//Balança de sólido 2
//Calculo peso com erro superior
PESO_ERRO_MAX_BLS2 := PRST_PESO_BLS2 + (PRST_PESO_BLS2 * (PRST_PORCENTAGEM_ERRO_PESO_BLS2 / 100));
//compara a banda
IF LEITURA_PESO_BLS2 > PESO_ERRO_MAX_BLS2 AND PRST_PESO_BLS2 > 0 AND BLS2_CARREGADA = TRUE AND BTS_PERMI_DESCAR_PESO_MAX_BLS2 = FALSE THEN
	AL_PESO_ALTO_BLS2 := TRUE;
ELSIF BTS_PERMI_DESCAR_PESO_MAX_BLS2 = TRUE OR PRST_PESO_BLS2 = 0 THEN	
	AL_PESO_ALTO_BLS2 := FALSE;	
END_IF

//Balança de sólido 3
//Calculo peso com erro superior
PESO_ERRO_MAX_BLS3 := PRST_PESO_BLS3 + (PRST_PESO_BLS3 * (PRST_PORCENTAGEM_ERRO_PESO_BLS3 / 100));
//compara a banda
IF LEITURA_PESO_BLS3 > PESO_ERRO_MAX_BLS3 AND PRST_PESO_BLS3 > 0 AND BLS3_CARREGADA = TRUE AND BTS_PERMI_DESCAR_PESO_MAX_BLS3 = FALSE THEN
	AL_PESO_ALTO_BLS3 := TRUE;
ELSIF BTS_PERMI_DESCAR_PESO_MAX_BLS3 = TRUE OR PRST_PESO_BLS3 = 0 THEN	
	AL_PESO_ALTO_BLS3 := FALSE;	
END_IF

//Balança de sólido 4
//Calculo peso com erro superior
PESO_ERRO_MAX_BLS4 := PRST_PESO_BLS4 + (PRST_PESO_BLS4 * (PRST_PORCENTAGEM_ERRO_PESO_BLS4 / 100));
//compara a banda
IF LEITURA_PESO_BLS4 > PESO_ERRO_MAX_BLS4 AND PRST_PESO_BLS4 > 0 AND BLS4_CARREGADA = TRUE AND BTS_PERMI_DESCAR_PESO_MAX_BLS4 = FALSE THEN
	AL_PESO_ALTO_BLS4 := TRUE;
ELSIF BTS_PERMI_DESCAR_PESO_MAX_BLS4 = TRUE OR PRST_PESO_BLS4 = 0 THEN	
	AL_PESO_ALTO_BLS4 := FALSE;	
END_IF

//Balança de sólido 5
//Calculo peso com erro superior
PESO_ERRO_MAX_BLS5 := PRST_PESO_BLS5 + (PRST_PESO_BLS5 * (PRST_PORCENTAGEM_ERRO_PESO_BLS5 / 100));
//compara a banda
IF LEITURA_PESO_BLS5 > PESO_ERRO_MAX_BLS5 AND PRST_PESO_BLS5 > 0 AND BLS5_CARREGADA = TRUE AND BTS_PERMI_DESCAR_PESO_MAX_BLS5 = FALSE THEN
	AL_PESO_ALTO_BLS5 := TRUE;
ELSIF BTS_PERMI_DESCAR_PESO_MAX_BLS5 = TRUE OR PRST_PESO_BLS5 = 0 THEN	
	AL_PESO_ALTO_BLS5 := FALSE;	
END_IF

//Balança de liquido 1
//Calculo peso com erro superior
PESO_ERRO_MAX_BLL1 := PRST_PESO_BLL1 + (PRST_PESO_BLL1 * (PRST_PORCENTAGEM_ERRO_PESO_BLL1 / 100));
//compara a banda
IF LEITURA_PESO_BLL1 > PESO_ERRO_MAX_BLL1 AND PRST_PESO_BLL1 > 0 AND BLL1_CARREGADA = TRUE AND BTS_PERMI_DESCAR_PESO_MAX_BLL1 = FALSE THEN
	AL_PESO_ALTO_BLL1 := TRUE;
ELSIF BTS_PERMI_DESCAR_PESO_MAX_BLL1 = TRUE OR PRST_PESO_BLL1 = 0 THEN	
	AL_PESO_ALTO_BLL1 := FALSE;	
END_IF

//Balança de liquido 2
//Calculo peso com erro superior
PESO_ERRO_MAX_BLL2 := PRST_PESO_BLL2 + (PRST_PESO_BLL2 * (PRST_PORCENTAGEM_ERRO_PESO_BLL2 / 100));
//compara a banda
IF LEITURA_PESO_BLL2 > PESO_ERRO_MAX_BLL2 AND PRST_PESO_BLL2 > 0 AND BLL2_CARREGADA = TRUE AND BTS_PERMI_DESCAR_PESO_MAX_BLL2 = FALSE THEN
	AL_PESO_ALTO_BLL2 := TRUE;
ELSIF BTS_PERMI_DESCAR_PESO_MAX_BLL2 = TRUE OR PRST_PESO_BLL2 = 0  THEN	
	AL_PESO_ALTO_BLL2 := FALSE;	
END_IF

//Balança de liquido 3
//Calculo peso com erro superior
PESO_ERRO_MAX_BLL3 := PRST_PESO_BLL3 + (PRST_PESO_BLL3 * (PRST_PORCENTAGEM_ERRO_PESO_BLL3 / 100));
//compara a banda
IF LEITURA_PESO_BLL3 > PESO_ERRO_MAX_BLL3 AND PRST_PESO_BLL3 > 0 AND BLL3_CARREGADA = TRUE AND BTS_PERMI_DESCAR_PESO_MAX_BLL3 = FALSE THEN
	AL_PESO_ALTO_BLL3 := TRUE;
ELSIF BTS_PERMI_DESCAR_PESO_MAX_BLL3 = TRUE OR PRST_PESO_BLL3 = 0  THEN	
	AL_PESO_ALTO_BLL3 := FALSE;	
END_IF

//Balança de liquido 4
//Calculo peso com erro superior
PESO_ERRO_MAX_BLL4 := PRST_PESO_BLL4 + (PRST_PESO_BLL4 * (PRST_PORCENTAGEM_ERRO_PESO_BLL4 / 100));
//compara a banda
IF LEITURA_PESO_BLL4 > PESO_ERRO_MAX_BLL4 AND PRST_PESO_BLL4 > 0 AND BLL4_CARREGADA = TRUE AND BTS_PERMI_DESCAR_PESO_MAX_BLL4 = FALSE THEN
	AL_PESO_ALTO_BLL4 := TRUE;
ELSIF BTS_PERMI_DESCAR_PESO_MAX_BLL4 = TRUE OR PRST_PESO_BLL4 = 0  THEN	
	AL_PESO_ALTO_BLL4 := FALSE;
END_IF

//======================= Exaustores =========================================================

//Alame estrela Exaustor FM2 

IF SD_EXFM2_E = TRUE AND (ED_CFEXFM2_P = FALSE AND ED_CFEXFM2_E = FALSE) THEN
	LIBERA_TEMPO_AL_FM2E:= TRUE;
ELSE
	LIBERA_TEMPO_AL_FM2E:= FALSE;
END_IF

TMR_TEMPO_ALARME_FM2_E(IN:= LIBERA_TEMPO_AL_FM2E, PT:= T#6S);

IF TMR_TEMPO_ALARME_FM2_E.Q = TRUE THEN
	AL_EXFM2_E:=TRUE;
END_IF

//Alame triangulo Exaustor FM2 

IF SD_EXFM2_T = TRUE AND (ED_CFEXFM2_P = FALSE AND ED_CFEXFM2_T = FALSE) THEN
	LIBERA_TEMPO_AL_FM2T:= TRUE;
ELSE
	LIBERA_TEMPO_AL_FM2T:= FALSE;
END_IF

TMR_TEMPO_ALARME_FM2_T(IN:= LIBERA_TEMPO_AL_FM2T, PT:= T#6S);

IF TMR_TEMPO_ALARME_FM2_T.Q = TRUE THEN
	AL_EXFM2_T:=TRUE;
END_IF

//Alame estrela Ventilador FM2 

IF SD_VEXFM2_E = TRUE AND (ED_CFVEXFM2_P = FALSE AND ED_CFVEXFM2_E = FALSE) THEN
	LIBERA_TEMPO_AL_VFM2E:= TRUE;
ELSE
	LIBERA_TEMPO_AL_VFM2E:= FALSE;
END_IF

TMR_TEMPO_ALARME_VFM2_E(IN:= LIBERA_TEMPO_AL_VFM2E, PT:= T#6S);

IF TMR_TEMPO_ALARME_VFM2_E.Q = TRUE THEN
	AL_VEXFM2_E:=TRUE;
END_IF

//Alame triangulo Ventilador FM2 

IF SD_VEXFM2_T = TRUE AND (ED_CFVEXFM2_P = FALSE AND ED_CFVEXFM2_T = FALSE) THEN
	LIBERA_TEMPO_AL_VFM2T:= TRUE;
ELSE
	LIBERA_TEMPO_AL_VFM2T:= FALSE;
END_IF

TMR_TEMPO_ALARME_VFM2_T(IN:= LIBERA_TEMPO_AL_VFM2T, PT:= T#6S);

IF TMR_TEMPO_ALARME_VFM2_T.Q = TRUE THEN
	AL_VEXFM2_T:=TRUE;
END_IF

//Alarme Exautor da torre (125 cv) 

IF ED_EX125_ALAR = TRUE THEN
	AL_EXTORRE:= TRUE;
END_IF


//Alarme ventilador do queimador (100 cv) 

IF ED_EX100_ALAR = TRUE THEN
	AL_VENTQUEIMADOR:= TRUE;
END_IF

//=============================== Bombas ============================================

//Alarme falta oleo bomba de alimentação 

IF SD_BAO = TRUE AND ED_NVBO = FALSE THEN
	LIBERA_TEMPO_AL_BALIOLEO := TRUE;
ELSE
	LIBERA_TEMPO_AL_BALIOLEO := FALSE;
END_IF

TMR_TEMPO_ALARME_BOMBA_ALIM_OLEO(IN:=LIBERA_TEMPO_AL_BALIOLEO, PT:=T#20S);

IF TMR_TEMPO_ALARME_BOMBA_ALIM_OLEO.Q = TRUE THEN
	AL_BOCOMBFALT := TRUE;
END_IF


//Bomba de Blend 
IF SD_BBD = TRUE AND ED_BB_D = FALSE THEN
	LIBERA_TEMPO_AL_BBBLEND:=TRUE;
ELSE
	LIBERA_TEMPO_AL_BBBLEND:= FALSE;
END_IF

TMR_TEMPO_ALARME_BBBLEND(IN:=LIBERA_TEMPO_AL_BBBLEND, PT:=T#15S);

IF TMR_TEMPO_ALARME_BBBLEND.Q = TRUE THEN
	AL_BBLEND:=TRUE;
END_IF


//Bomba de Silicato (Acrilato) 
IF SD_BSIL = TRUE AND ED_BSI_D = FALSE THEN
	LIBERA_TEMPO_AL_BBSILICATO:=TRUE;
ELSE
	LIBERA_TEMPO_AL_BBSILICATO:= FALSE;
END_IF

TMR_TEMPO_ALARME_BBSILICATO(IN:=LIBERA_TEMPO_AL_BBSILICATO, PT:=T#15S);

IF TMR_TEMPO_ALARME_BBSILICATO.Q = TRUE THEN
	AL_SILI:=TRUE;
END_IF


//Bomba de Sulfonico 
IF SD_BSUL = TRUE AND ED_BSU_D = FALSE THEN
	LIBERA_TEMPO_AL_BBSULFONICO:=TRUE;
ELSE
	LIBERA_TEMPO_AL_BBSULFONICO:= FALSE;
END_IF

TMR_TEMPO_ALARME_BBSULFONICO(IN:=LIBERA_TEMPO_AL_BBSULFONICO, PT:=T#15S);

IF TMR_TEMPO_ALARME_BBSULFONICO.Q = TRUE THEN
	AL_BBSULFONICO:=TRUE;
END_IF


//Bomba de Agua 
IF SD_BAG = TRUE AND ED_BA_D = FALSE THEN
	LIBERA_TEMPO_AL_BBAGUA:=TRUE;
ELSE
	LIBERA_TEMPO_AL_BBAGUA:= FALSE;
END_IF

TMR_TEMPO_ALARME_BBAGUA(IN:=LIBERA_TEMPO_AL_BBAGUA, PT:=T#15S);

IF TMR_TEMPO_ALARME_BBAGUA.Q = TRUE THEN
	AL_BBAGUA:=TRUE;
END_IF


//Bomba de Soda 
IF SD_BSOD = TRUE AND ED_BSO_D = FALSE THEN
	LIBERA_TEMPO_AL_BBSODA:=TRUE;
ELSE
	LIBERA_TEMPO_AL_BBSODA:= FALSE;
END_IF

TMR_TEMPO_ALARME_BBSODA(IN:=LIBERA_TEMPO_AL_BBSODA, PT:=T#15S);

IF TMR_TEMPO_ALARME_BBSODA.Q = TRUE THEN
	AL_BBSODA:=TRUE;
END_IF


//Bomba de Transferencia
IF SD_BBTRANS = TRUE AND ED_BTRA_D = FALSE THEN
	LIBERA_TEMPO_AL_BBTRANSFE:=TRUE;
ELSE
	LIBERA_TEMPO_AL_BBTRANSFE:= FALSE;
END_IF

TMR_BBTRANSFERENCIA_ALARME(IN:=LIBERA_TEMPO_AL_BBTRANSFE, PT:=T#15S);

IF TMR_BBTRANSFERENCIA_ALARME.Q = TRUE THEN
	AL_BBTRANS:=TRUE;
END_IF


//Bomba de Baixa
IF SD_BB = TRUE AND ED_BB_F = TRUE THEN
	AL_BB := TRUE;
END_IF

//Bomba de alta 1
IF SD_BA1 = TRUE AND ED_BA1_F = TRUE THEN
	AL_BA1 := TRUE;
END_IF

//Bomba de alta 2
IF SD_BA2 = TRUE AND ED_BA2_F = TRUE THEN
	AL_BA2 := TRUE;
END_IF

//Falha de pressão Bomba alta 1
IF SD_BA1 = TRUE AND ED_PRTBA1 = TRUE THEN
	LIBERA_TEMPO_AL_FALHA_PRESSAO_BBALTA1:=TRUE;
ELSE
	LIBERA_TEMPO_AL_FALHA_PRESSAO_BBALTA1:= FALSE;
END_IF

TMR_FALHA_PRESSAO_BBALTA1_ALARME(IN:=LIBERA_TEMPO_AL_FALHA_PRESSAO_BBALTA1, PT:=T#15S);

IF TMR_FALHA_PRESSAO_BBALTA1_ALARME.Q = TRUE THEN
	AL_FPBA1:=TRUE;
END_IF

//Falha de pressão Bomba alta 2
IF SD_BA2 = TRUE AND ED_PRTBA2 = TRUE THEN
	LIBERA_TEMPO_AL_FALHA_PRESSAO_BBALTA2:=TRUE;
ELSE
	LIBERA_TEMPO_AL_FALHA_PRESSAO_BBALTA2:= FALSE;
END_IF

TMR_FALHA_PRESSAO_BBALTA2_ALARME(IN:=LIBERA_TEMPO_AL_FALHA_PRESSAO_BBALTA2, PT:=T#15S);

IF TMR_FALHA_PRESSAO_BBALTA2_ALARME.Q = TRUE THEN
	AL_FPBA2:=TRUE;
END_IF

(*===================================== Moinho =====================================

//Alame triangulo 

IF SD_MH_T = TRUE AND (ED_CFMH_P = FALSE OR ED_CFMH_T = FALSE) THEN
	LIBERA_TEMPO_AL_TRIAN_MOINHO:= TRUE;
ELSE
	LIBERA_TEMPO_AL_TRIAN_MOINHO:= FALSE;
END_IF

TMR_TRIANGULO_MOINHO_ALARME(IN:= LIBERA_TEMPO_AL_TRIAN_MOINHO, PT:= T#6S);

IF TMR_TRIANGULO_MOINHO_ALARME.Q = TRUE THEN
	AL_MHT := TRUE;
END_IF

//Alame estrela 

IF SD_MH_E = TRUE AND (ED_CFMH_P = FALSE OR ED_CFMH_E = FALSE) THEN
	LIBERA_TEMPO_AL_ESTRELA_MOINHO:= TRUE;
ELSE
	LIBERA_TEMPO_AL_ESTRELA_MOINHO:= FALSE;
END_IF

TMR_ESTRELA_MOINHO_ALARME(IN:= LIBERA_TEMPO_AL_ESTRELA_MOINHO, PT:= T#6S);

IF TMR_ESTRELA_MOINHO_ALARME.Q = TRUE THEN
	AL_MHE := TRUE;
END_IF*)

//==================================== Esteiras =====================================

//Alame esteira TC8 não entrou  

IF SD_ESTTC8 = TRUE AND NOT ED_ESTTC8_D  THEN
	LIBERA_TEMPO_AL_TC8:= TRUE;
ELSE
	LIBERA_TEMPO_AL_TC8:= FALSE;
END_IF

TMR_TEMPO_ALARME_ESTTC8(IN:= LIBERA_TEMPO_AL_TC8, PT:= T#5S);

IF TMR_TEMPO_ALARME_ESTTC8.Q THEN
	AL_ESTTC8:=TRUE;
END_IF

//Esteira saida Torre  

IF SD_ESTSTORRE = TRUE AND ED_ESTST_L = FALSE THEN
	LIBERA_TEMPO_AL_ESTSTORRE:=TRUE;
ELSE	
	LIBERA_TEMPO_AL_ESTSTORRE:=FALSE;
END_IF

T_Alarme_ESTSTORRE(IN:= LIBERA_TEMPO_AL_ESTSTORRE, PT:= T#5S);

IF T_Alarme_ESTSTORRE.Q = TRUE THEN
	AL_ESTSAITORRE:=TRUE;
END_IF
//================================== Peneiras ========================================

// Peneira 1
IF SD_M1PN = TRUE AND ED_PNM1_L = FALSE  THEN
	LIBERA_TEMPO_AL_PN1:= TRUE;
ELSE
	LIBERA_TEMPO_AL_PN1:= FALSE;
END_IF

TMR_TEMPO_ALARME_PN1(IN:= LIBERA_TEMPO_AL_PN1, PT:= T#5S);

IF TMR_TEMPO_ALARME_PN1.Q THEN
	AL_PN1:=TRUE;
END_IF

// Peneira 2
IF SD_M2PN = TRUE AND  ED_PNM2_L = FALSE  THEN
	LIBERA_TEMPO_AL_PN2:= TRUE;
ELSE
	LIBERA_TEMPO_AL_PN2:= FALSE;
END_IF

TMR_TEMPO_ALARME_PN2(IN:= LIBERA_TEMPO_AL_PN2, PT:= T#5S);

IF TMR_TEMPO_ALARME_PN2.Q THEN
	AL_PN2:=TRUE;
END_IF

// Peneira 3
IF SD_M3PN = TRUE AND ED_PNM3_L = FALSE  THEN
	LIBERA_TEMPO_AL_PN3:= TRUE;
ELSE
	LIBERA_TEMPO_AL_PN3:= FALSE;
END_IF

TMR_TEMPO_ALARME_PN3(IN:= LIBERA_TEMPO_AL_PN3, PT:= T#5S);

IF TMR_TEMPO_ALARME_PN3.Q THEN
	AL_PN3:=TRUE;
END_IF

// Peneira 4
IF SD_M4PN = TRUE AND ED_PNM4_L = FALSE  THEN
	LIBERA_TEMPO_AL_PN4:= TRUE;
ELSE
	LIBERA_TEMPO_AL_PN4:= FALSE;
END_IF

TMR_TEMPO_ALARME_PN4(IN:= LIBERA_TEMPO_AL_PN4, PT:= T#5S);

IF TMR_TEMPO_ALARME_PN4.Q THEN
	AL_PN4:=TRUE;
END_IF

//Elevador 2 ==========================================================================

IF SD_EL2 AND NOT ED_EL2_L THEN
	LIBERA_TEMPO_AL_EL2:=TRUE;
ELSE	
	LIBERA_TEMPO_AL_EL2:=FALSE;
END_IF

T_Alarme_EL2(IN:= LIBERA_TEMPO_AL_EL2, PT:= T#5S);

IF T_Alarme_EL2.Q THEN
	AL_EL2:=TRUE;
END_IF



//Air Lift ===========================================================================

IF ED_AIRLFT_F = TRUE THEN
	AL_AIRLF:= TRUE;
END_IF


//Queimador ===========================================================================

IF ED_PROGFOR_ALAR = TRUE THEN
	AL_QUEIMADOR := TRUE;
END_IF

//Alarme alta temperatura torre ==============================================
IF TEMP_TORRE > PRST_SEGURANCA_TORRE AND SILENCIA_AL_ALTA_TEMPE_TORRE = FALSE THEN
	AL_ALTA_TEMPE_TORRE := TRUE;
ELSE
	AL_ALTA_TEMPE_TORRE := FALSE;
END_IF

//Silencia alarme
IF TEMP_TORRE < PRST_SEGURANCA_TORRE  THEN
	SILENCIA_AL_ALTA_TEMPE_TORRE := FALSE;
END_IF

//Alarme Sonoro =======================================================================

IF AL_ALTA_TEMPE_TORRE = TRUE THEN
	SD_SONORO := TRUE;
ELSE
	SD_SONORO := FALSE;
END_IF

//Dosadoras Schenck ===================================================================

//Y08 Comm.-Error Host  (Erro de Comunicação) ==================================

//DS01 - PB01
IF %QX21752.5 = TRUE THEN
	AL_SY08COMM_ERRORHOST_DS01 := TRUE;
ELSE
	AL_SY08COMM_ERRORHOST_DS01 := FALSE;
END_IF

//DS02
IF %QX21808.5 = TRUE THEN
	AL_SY08COMM_ERRORHOST_DS02 := TRUE;
ELSE
	AL_SY08COMM_ERRORHOST_DS02 := FALSE;
END_IF

//DS03
IF %QX21864.5 = TRUE THEN
	AL_SY08COMM_ERRORHOST_DS03 := TRUE;
ELSE
	AL_SY08COMM_ERRORHOST_DS03 := FALSE;
END_IF

//DS04
IF %QX21920.5 = TRUE THEN
	AL_SY08COMM_ERRORHOST_DS04 := TRUE;
ELSE
	AL_SY08COMM_ERRORHOST_DS04 := FALSE;
END_IF

//DS05
IF %QX21976.5 = TRUE THEN
	AL_SY08COMM_ERRORHOST_DS05 := TRUE;
ELSE
	AL_SY08COMM_ERRORHOST_DS05 := FALSE;
END_IF

//DS07
IF %QX22032.5 = TRUE THEN
	AL_SY08COMM_ERRORHOST_DS07 := TRUE;
ELSE
	AL_SY08COMM_ERRORHOST_DS07 := FALSE;
END_IF

//DS08
IF %QX22144.5 = TRUE THEN
	AL_SY08COMM_ERRORHOST_DS08 := TRUE;
ELSE
	AL_SY08COMM_ERRORHOST_DS08 := FALSE;
END_IF
	
//DS09
IF %QX22088.5 = TRUE THEN
	AL_SY08COMM_ERRORHOST_DS09 := TRUE;
ELSE
	AL_SY08COMM_ERRORHOST_DS09 := FALSE;
END_IF

//DS10
IF %QX22200.5 = TRUE THEN
	AL_SY08COMM_ERRORHOST_DS10 := TRUE;
ELSE
	AL_SY08COMM_ERRORHOST_DS10 := FALSE;
END_IF

//DS11 - PB11
IF %QX22256.5 = TRUE THEN
	AL_SY08COMM_ERRORHOST_DS11 := TRUE;
ELSE
	AL_SY08COMM_ERRORHOST_DS11 := FALSE;
END_IF

//DS12
IF %QX22312.5 = TRUE THEN
	AL_SY08COMM_ERRORHOST_DS12 := TRUE;
ELSE
	AL_SY08COMM_ERRORHOST_DS12 := FALSE;
END_IF

//DSTORRE
IF %QX22368.5 = TRUE THEN
	AL_SY08COMM_ERRORHOST_DSTORRE := TRUE;
ELSE
	AL_SY08COMM_ERRORHOST_DSTORRE := FALSE;
END_IF


//SC05 External Event1 (Falha acionamento Inversor) ==================================

//DS01 - PB01
IF %IX15385.4 = TRUE THEN
	AL_SC05EXTERNAL_EVENT_DS01 := TRUE;
ELSE
	AL_SC05EXTERNAL_EVENT_DS01 := FALSE;
END_IF

//DS02
IF %IX15387.4 = TRUE THEN
	AL_SC05EXTERNAL_EVENT_DS02 := TRUE;
ELSE
	AL_SC05EXTERNAL_EVENT_DS02 := FALSE;
END_IF

//DS03
IF %IX15389.4 = TRUE THEN
	AL_SC05EXTERNAL_EVENT_DS03 := TRUE;
ELSE
	AL_SC05EXTERNAL_EVENT_DS03 := FALSE;
END_IF

//DS04
IF %IX15391.4 = TRUE THEN
	AL_SC05EXTERNAL_EVENT_DS04 := TRUE;
ELSE
	AL_SC05EXTERNAL_EVENT_DS04 := FALSE;
END_IF

//DS05
IF %IX15393.4 = TRUE THEN
	AL_SC05EXTERNAL_EVENT_DS05 := TRUE;
ELSE
	AL_SC05EXTERNAL_EVENT_DS05 := FALSE;
END_IF

//DS07
IF %IX15395.4 = TRUE THEN
	AL_SC05EXTERNAL_EVENT_DS07 := TRUE;
ELSE
	AL_SC05EXTERNAL_EVENT_DS07 := FALSE;
END_IF

//DS08
IF %IX15397.4 = TRUE THEN
	AL_SC05EXTERNAL_EVENT_DS08 := TRUE;
ELSE
	AL_SC05EXTERNAL_EVENT_DS08 := FALSE;
END_IF
	
//DS09
IF %IX15399.4 = TRUE THEN
	AL_SC05EXTERNAL_EVENT_DS09 := TRUE;
ELSE
	AL_SC05EXTERNAL_EVENT_DS09 := FALSE;
END_IF

//DS10
IF %IX15401.4 = TRUE THEN
	AL_SC05EXTERNAL_EVENT_DS10 := TRUE;
ELSE
	AL_SC05EXTERNAL_EVENT_DS10 := FALSE;
END_IF

//DS11 - PB11
IF %IX15403.4 = TRUE THEN
	AL_SC05EXTERNAL_EVENT_DS11 := TRUE;
ELSE
	AL_SC05EXTERNAL_EVENT_DS11 := FALSE;
END_IF

//DS12
IF %IX15405.4 = TRUE THEN
	AL_SC05EXTERNAL_EVENT_DS12 := TRUE;
ELSE
	AL_SC05EXTERNAL_EVENT_DS12 := FALSE;
END_IF

//DSTORRE
IF %IX15407.4 = TRUE THEN
	AL_SC05EXTERNAL_EVENT_DSTORRE := TRUE;
ELSE
	AL_SC05EXTERNAL_EVENT_DSTORRE := FALSE;
END_IF

//SC09 Feedback Gate  DS01 (Confirmação Valvula Fechada) ==================================

//DS01 - PB01
IF %IX15384.0 = TRUE THEN
	AL_SC09FEEDDBACK_GATE_DS01 := TRUE;
ELSE
	AL_SC09FEEDDBACK_GATE_DS01 := FALSE;
END_IF

//DS02
IF %IX15386.0 = TRUE THEN
	AL_SC09FEEDDBACK_GATE_DS02 := TRUE;
ELSE
	AL_SC09FEEDDBACK_GATE_DS02 := FALSE;
END_IF

//DS03
IF %IX15388.0 = TRUE THEN
	AL_SC09FEEDDBACK_GATE_DS03 := TRUE;
ELSE
	AL_SC09FEEDDBACK_GATE_DS03 := FALSE;
END_IF

//DS04
IF %IX15390.0 = TRUE THEN
	AL_SC09FEEDDBACK_GATE_DS04 := TRUE;
ELSE
	AL_SC09FEEDDBACK_GATE_DS04 := FALSE;
END_IF

//DS05
IF %IX15392.0 = TRUE THEN
	AL_SC09FEEDDBACK_GATE_DS05 := TRUE;
ELSE
	AL_SC09FEEDDBACK_GATE_DS05 := FALSE;
END_IF

//DS07
IF %IX15394.0 = TRUE THEN
	AL_SC09FEEDDBACK_GATE_DS07 := TRUE;
ELSE
	AL_SC09FEEDDBACK_GATE_DS07 := FALSE;
END_IF

//DS08
IF %IX15396.0 = TRUE THEN
	AL_SC09FEEDDBACK_GATE_DS08 := TRUE;
ELSE
	AL_SC09FEEDDBACK_GATE_DS08 := FALSE;
END_IF
	
//DS09
IF %IX15398.0 = TRUE THEN
	AL_SC09FEEDDBACK_GATE_DS09 := TRUE;
ELSE
	AL_SC09FEEDDBACK_GATE_DS09 := FALSE;
END_IF

//DS10
IF %IX15400.0 = TRUE THEN
	AL_SC09FEEDDBACK_GATE_DS10 := TRUE;
ELSE
	AL_SC09FEEDDBACK_GATE_DS10 := FALSE;
END_IF

//DS11 - PB11
IF %IX15402.0 = TRUE THEN
	AL_SC09FEEDDBACK_GATE_DS11 := TRUE;
ELSE
	AL_SC09FEEDDBACK_GATE_DS11 := FALSE;
END_IF

//DS12
IF %IX15404.0 = TRUE THEN
	AL_SC09FEEDDBACK_GATE_DS12 := TRUE;
ELSE
	AL_SC09FEEDDBACK_GATE_DS12 := FALSE;
END_IF

//DSTORRE
IF %IX15406.0 = TRUE THEN
	AL_SC09FEEDDBACK_GATE_DSTORRE := TRUE;
ELSE
	AL_SC09FEEDDBACK_GATE_DSTORRE := FALSE;
END_IF

//HI05 Control Deviation DS01 (Controle de Desvio) ==================================

//DS01 - PB01
IF %IX15409.4 = TRUE THEN
	AL_HI05_CONTROL_DEVIATION_DS01 := TRUE;
ELSE
	AL_HI05_CONTROL_DEVIATION_DS01 := FALSE;
END_IF

//DS02
IF %IX15411.4 = TRUE THEN
	AL_HI05_CONTROL_DEVIATION_DS02 := TRUE;
ELSE
	AL_HI05_CONTROL_DEVIATION_DS02 := FALSE;
END_IF

//DS03
IF %IX15413.4 = TRUE THEN
	AL_HI05_CONTROL_DEVIATION_DS03 := TRUE;
ELSE
	AL_HI05_CONTROL_DEVIATION_DS03 := FALSE;
END_IF

//DS04
IF %IX15415.4 = TRUE THEN
	AL_HI05_CONTROL_DEVIATION_DS04 := TRUE;
ELSE
	AL_HI05_CONTROL_DEVIATION_DS04 := FALSE;
END_IF

//DS05
IF %IX15417.4 = TRUE THEN
	AL_HI05_CONTROL_DEVIATION_DS05 := TRUE;
ELSE
	AL_HI05_CONTROL_DEVIATION_DS05 := FALSE;
END_IF

//DS07
IF %IX15419.4 = TRUE THEN
	AL_HI05_CONTROL_DEVIATION_DS07 := TRUE;
ELSE
	AL_HI05_CONTROL_DEVIATION_DS07 := FALSE;
END_IF

//DS08
IF %IX15421.4 = TRUE THEN
	AL_HI05_CONTROL_DEVIATION_DS08 := TRUE;
ELSE
	AL_HI05_CONTROL_DEVIATION_DS08 := FALSE;
END_IF
	
//DS09
IF %IX15423.4 = TRUE THEN
	AL_HI05_CONTROL_DEVIATION_DS09 := TRUE;
ELSE
	AL_HI05_CONTROL_DEVIATION_DS09 := FALSE;
END_IF

//DS10
IF %IX15425.4 = TRUE THEN
	AL_HI05_CONTROL_DEVIATION_DS10 := TRUE;
ELSE
	AL_HI05_CONTROL_DEVIATION_DS10 := FALSE;
END_IF

//DS11 - PB11
IF %IX15427.4 = TRUE THEN
	AL_HI05_CONTROL_DEVIATION_DS11 := TRUE;
ELSE
	AL_HI05_CONTROL_DEVIATION_DS11 := FALSE;
END_IF

//DS12
IF %IX15429.4 = TRUE THEN
	AL_HI05_CONTROL_DEVIATION_DS12 := TRUE;
ELSE
	AL_HI05_CONTROL_DEVIATION_DS12 := FALSE;
END_IF

//DS14
IF %IX15431.4 = TRUE THEN
	AL_HI05_CONTROL_DEVIATION_DS14 := TRUE;
ELSE
	AL_HI05_CONTROL_DEVIATION_DS14 := FALSE;
END_IF

//DSTORRE
IF %IX15431.4 = TRUE THEN
	AL_HI05_CONTROL_DEVIATION_DSTORRE := TRUE;
ELSE
	AL_HI05_CONTROL_DEVIATION_DSTORRE := FALSE;
END_IF


//SIRENE AUDIO VISUAL ALARME DOSADORES - ROBY 07/02/22 - INICIO
//===================================================================
IF (BTS_MAPH1 = TRUE OR BTS_MAPH2 = TRUE) AND (AL_HI05_CONTROL_DEVIATION_DS01 = TRUE OR AL_HI05_CONTROL_DEVIATION_DS02 = TRUE OR 
AL_HI05_CONTROL_DEVIATION_DS03 = TRUE OR AL_HI05_CONTROL_DEVIATION_DS04 = TRUE OR 
AL_HI05_CONTROL_DEVIATION_DS05 = TRUE  OR AL_HI05_CONTROL_DEVIATION_DS12 = TRUE OR 
AL_HI05_CONTROL_DEVIATION_DS08 = TRUE OR AL_HI05_CONTROL_DEVIATION_DS09 = TRUE OR 
AL_HI05_CONTROL_DEVIATION_DS10 = TRUE OR AL_HI05_CONTROL_DEVIATION_DS11 = TRUE OR 
AL_HI05_CONTROL_DEVIATION_DSTORRE = TRUE OR AL_HI05_CONTROL_DEVIATION_DS07 = TRUE OR
AL_HI05_CONTROL_DEVIATION_DS14 = TRUE) THEN
LIBERA_TEMP_AL_SIR_DOSADORES := TRUE;
ELSE
	LIBERA_TEMP_AL_SIR_DOSADORES := FALSE;
		AL_SIR_DOSADORES:=FALSE;

END_IF
TEMP_AL_SIR_DOSADORES(IN:= LIBERA_TEMP_AL_SIR_DOSADORES, PT:= T#10S);

IF TEMP_AL_SIR_DOSADORES.Q = TRUE THEN
	BLINK_SIRENE(ENABLE:= TRUE, TIMELOW:= T#10S, TIMEHIGH:= T#1S, OUT=> AL_SIR_DOSADORES);
END_IF
//==============================================================

//SIRENE AUDIO VISUAL ALARME DOSADORES - ROBY 07/02/22 - FIM

//INICIO MUDA PH1 PARA MANUAL CASO PERSISTA POR MAIS DE 30S O ALARME DE DESVIO DOS DOSADORES.

IF BTS_MAPH1 = TRUE AND (AL_HI05_CONTROL_DEVIATION_DS01 = TRUE OR AL_HI05_CONTROL_DEVIATION_DS05 = TRUE OR AL_HI05_CONTROL_DEVIATION_DS04 = TRUE OR 
AL_HI05_CONTROL_DEVIATION_DS03 = TRUE OR AL_HI05_CONTROL_DEVIATION_DS02 = TRUE) THEN
BTS_MAPH1 := FALSE;
END_IF

//FIM MUDA PH1 PARA MANUAL CASO PERSISTA POR MAIS DE 30S O ALARME DE DESVIO DOS DOSADORES.
	

//INICIO MUDA PH2 PARA MANUAL CASO PERSISTA POR MAIS DE 30S O ALARME DE DESVIO DOS DOSADORES.

IF BTS_MAPH2 = TRUE AND (AL_HI05_CONTROL_DEVIATION_DS12 = TRUE OR AL_HI05_CONTROL_DEVIATION_DS08 = TRUE OR AL_HI05_CONTROL_DEVIATION_DS09 = TRUE OR 
AL_HI05_CONTROL_DEVIATION_DS10 = TRUE OR AL_HI05_CONTROL_DEVIATION_DS11 = TRUE) THEN
BTS_MAPH2 := FALSE;
END_IF

//FIM MUDA PH2 PARA MANUAL CASO PERSISTA POR MAIS DE 30S O ALARME DE DESVIO DOS DOSADORES.



// Reset dos alarmes ==================================================================	
// Reset dos alarmes ==================================================================

IF BTS_RSTAL = TRUE THEN
	AL_SIR_DOSADORES:=FALSE;
	AL_EXTORRE := FALSE;
	AL_VENTQUEIMADOR := FALSE;
	AL_BOCOMBFALT := FALSE;
	AL_EXFM2_E := FALSE;
	AL_EXFM2_T := FALSE;
	AL_VEXFM2_E := FALSE;
	AL_VEXFM2_T := FALSE;
	AL_ESTTC8 := FALSE;
	AL_PN1 := FALSE;
	AL_PN2 := FALSE;
	AL_PN3 := FALSE;
	AL_PN4 := FALSE;
	AL_EL2 := FALSE;
	AL_ESTSAIRLF := FALSE;
	AL_AIRLF := FALSE;
	AL_ESTSAITORRE := FALSE;
	AL_QUEIMADOR := FALSE;
	AL_RPO1 := FALSE;
	AL_RPO2 := FALSE;
	AL_RPO3 := FALSE;
	AL_RPO4 := FALSE;
	AL_RPO5 := FALSE;
	AL_RC6H := FALSE;
	AL_RC7I := FALSE;
	AL_BLS1D := FALSE;
	AL_BLS2D := FALSE;
	AL_BLS3D := FALSE;
	AL_BLS4D := FALSE;
	AL_BLS5D := FALSE;
	AL_BL1D := FALSE;
	AL_BL2D := FALSE;
	AL_BL3D := FALSE;
	AL_BL4D := FALSE;
	AL_BLL1L := FALSE;
	AL_BLL2L := FALSE;
	AL_BLL3L := FALSE;
	AL_BLL4L := FALSE;
	AL_BLL1R := FALSE;
	AL_BLL2R := FALSE;
	AL_BLL3R := FALSE;
	AL_BLL4R := FALSE;
	AL_BBLEND := FALSE;
	AL_SILI := FALSE;
	AL_BBSULFONICO := FALSE;
	AL_BBAGUA := FALSE;
	AL_BBSODA := FALSE;
	AL_BB := FALSE;
	AL_BA1 := FALSE;
	AL_BA2 := FALSE;
	AL_FPBA1 := FALSE;
	AL_FPBA2 := FALSE;
	AL_MHT := FALSE;
	AL_MHE := FALSE;
	AL_ALTA_TEMPE_TORRE := FALSE;
	SILENCIA_AL_ALTA_TEMPE_TORRE := TRUE;
	
	BTS_RSTAL := FALSE;
	
	
	


END_IF
//=========================================================================
	//             transferencia para região de comunicação com supervisório
	//=========================================================================1
BLINK_ALARMES(ENABLE:= TRUE, TIMELOW:= T#2S, TIMEHIGH:= T#2S, OUT=> ATUALIZA_ALARMES);
IF ATUALIZA_ALARMES = TRUE OR BTS_RSTAL = TRUE THEN
		%QX3151.0 := AL_RPO1;
	%QX3151.1 := AL_RPO2;
	%QX3151.2 :=  AL_RPO3;
	%QX3151.3 := AL_RPO4;
	%QX3151.4 := AL_RPO5;
	%QX3151.5 := AL_RC6H;
	%QX3151.6 := AL_RC7I;
	%QX3151.7 := AL_BLS1D;
	%QX3150.0 := AL_BLS2D;
	%QX3150.1 := AL_BLS3D;
	%QX3150.2 := AL_BLS4D;
	%QX3150.3 := AL_BLS5D;
	%QX3150.4 := AL_BL1D;
	%QX3150.5 := AL_BL2D;
	%QX3150.6 := AL_BL3D;
	%QX3150.7 := AL_BL4D;
	%QX3153.0 := AL_BLL1R;
	%QX3153.1 := AL_BLL1L;
	%QX3153.2 := AL_BLL2R;
	%QX3153.3 := AL_BLL2L;
	%QX3153.4 := AL_BLL3R;
	%QX3153.5 := AL_BLL3L;
	%QX3153.6 := AL_BLL4R;
	%QX3153.7 := AL_BLL4L;
	%QX3152.0 := AL_CFMXP;
	%QX3152.1 := AL_MXE;
	%QX3152.2 := AL_BOCOMB;
	%QX3152.3 := AL_BDP;
	%QX3152.4 := AL_BB;
	%QX3152.5 := AL_BA1;
	%QX3152.6 := AL_BA2;
	%QX3155.0 := AL_MHE;
	%QX3155.1 := AL_EXFM1_E;
	%QX3155.2 := AL_EXFM2;
	%QX3155.3 := AL_EXFM3;
	%QX3155.4 := AL_TC3;
	%QX3155.5 := AL_ESTSAIRLF;
	%QX3155.6 := AL_AIRLF;
	%QX3155.7 := AL_EL2;
	%QX3154.0 := AL_ESTTC8;
	%QX3154.1 := AL_FPBA1;
	%QX3154.2 := AL_FPBA2;
	%QX3154.3 := AL_MHT;
	%QX3154.4 := AL_VLRNA;
	%QX3154.5 := AL_VLRNF;
	%QX3154.6 := AL_BBTRANS;
	%QX3154.7 := AL_EXFM1_T;
	%QX3157.0 := AL_BBLEND;
	%QX3157.1 := AL_SILI;
	%QX3157.2 := AL_EXTORRE;
	%QX3157.3 := AL_GERAL;
	%QX3157.4 := AL_VENTQUEIMADOR;
	%QX3157.5 := AL_BOCOMBFALT;
	%QX3157.6 := AL_EXFM2_E;
	%QX3157.7 := AL_EXFM2_T;
	%QX3156.0 := AL_VEXFM2_E;
	%QX3156.1 := AL_VEXFM2_T;
	%QX3156.2 := AL_PN1;
	%QX3156.3 := AL_PN2;
	%QX3156.4 := AL_PN3;
	%QX3156.5 := AL_PN4;
	%QX3156.6 := AL_ESTSAITORRE;
	%QX3156.7 := AL_DESCARGA_BLS1;
	%QX3159.0 := AL_DESCARGA_BLS2;
	%QX3159.1 := AL_DESCARGA_BLS3;
	%QX3159.2 := AL_DESCARGA_BLS4;
	%QX3159.3 := AL_DESCARGA_BLS5;
	%QX3159.4 := AL_DESCARGA_BLL1;
	%QX3159.5 := AL_DESCARGA_BLL2;
	%QX3159.6 := AL_DESCARGA_BLL3;
	%QX3159.7 := AL_DESCARGA_BLL4;
	%QX3158.0 := AL_QUEIMADOR;
	%QX3158.1 := AL_BBSULFONICO;
	%QX3158.2 := AL_BBAGUA;
	%QX3158.3 := AL_BBSODA;
	%QX3158.4 := AL_PESO_ALTO_BLS1;
	%QX3158.5 := AL_PESO_ALTO_BLS2;
	%QX3158.6 := AL_PESO_ALTO_BLS3;
	%QX3158.7 := AL_PESO_ALTO_BLS4;
	%QX3161.0 := AL_PESO_ALTO_BLS5;
	%QX3161.1 := AL_PESO_ALTO_BLL1;
	%QX3161.2 := AL_PESO_ALTO_BLL2;
	%QX3161.3 := AL_PESO_ALTO_BLL3;
	%QX3161.4 := AL_PESO_ALTO_BLL4;
	%QX3161.5 := AL_ALTA_TEMPE_TORRE;
	%QX3161.6 := AL_SY08COMM_ERRORHOST_DS01;
	%QX3161.7 := AL_SY08COMM_ERRORHOST_DS02;
	%QX3160.0 := AL_SY08COMM_ERRORHOST_DS03;
	%QX3160.1 := AL_SY08COMM_ERRORHOST_DS04;
	%QX3160.2 := AL_SY08COMM_ERRORHOST_DS05;
	%QX3160.3 := AL_SY08COMM_ERRORHOST_DS07;
	%QX3160.4 := AL_SY08COMM_ERRORHOST_DS08;
	%QX3160.5 := AL_SY08COMM_ERRORHOST_DS09;
	%QX3160.6 := AL_SY08COMM_ERRORHOST_DS10;
	%QX3160.7 := AL_SY08COMM_ERRORHOST_DS11;
	%QX3163.0 := AL_SY08COMM_ERRORHOST_DS12;
	%QX3170.0 := AL_SY08COMM_ERRORHOST_DS14; // Verificar
	%QX3163.1 := AL_SY08COMM_ERRORHOST_DSTORRE;
	%QX3163.2 := AL_SC05EXTERNAL_EVENT_DS01;
	%QX3163.3 := AL_SC05EXTERNAL_EVENT_DS02;
	%QX3163.4 := AL_SC05EXTERNAL_EVENT_DS03;
	%QX3163.5 := AL_SC05EXTERNAL_EVENT_DS04;
	%QX3163.6 := AL_SC05EXTERNAL_EVENT_DS05;
	%QX3163.7 := AL_SC05EXTERNAL_EVENT_DS07;
	%QX3162.0 := AL_SC05EXTERNAL_EVENT_DS08;
	%QX3162.1 := AL_SC05EXTERNAL_EVENT_DS09;
	%QX3162.2 := AL_SC05EXTERNAL_EVENT_DS10;
	%QX3162.3 := AL_SC05EXTERNAL_EVENT_DS11;
	%QX3162.4 := AL_SC05EXTERNAL_EVENT_DS12;
	%QX3170.1 := AL_SC05EXTERNAL_EVENT_DS14; // Verificar
	%QX3162.5 := AL_SC05EXTERNAL_EVENT_DSTORRE;
	%QX3162.6 := AL_SC09FEEDDBACK_GATE_DS01;
	%QX3162.7 := AL_SC09FEEDDBACK_GATE_DS02;
	%QX3165.0 := AL_SC09FEEDDBACK_GATE_DS03;
	%QX3165.1 := AL_SC09FEEDDBACK_GATE_DS04;
	%QX3165.2 := AL_SC09FEEDDBACK_GATE_DS05;
	%QX3165.3 := AL_SC09FEEDDBACK_GATE_DS07;
	%QX3165.4 := AL_SC09FEEDDBACK_GATE_DS08;
	%QX3165.5 := AL_SC09FEEDDBACK_GATE_DS09;
	%QX3165.6 := AL_SC09FEEDDBACK_GATE_DS10;
	%QX3165.7 := AL_SC09FEEDDBACK_GATE_DS11;
	%QX3164.0 := AL_SC09FEEDDBACK_GATE_DS12;
	%QX3170.2 := AL_SC09FEEDDBACK_GATE_DS14; // Verificar
	%QX3164.1 := AL_SC09FEEDDBACK_GATE_DSTORRE;
	%QX3164.2 := AL_HI05_CONTROL_DEVIATION_DS01;
	%QX3164.3 := AL_HI05_CONTROL_DEVIATION_DS02;
	%QX3164.4 := AL_HI05_CONTROL_DEVIATION_DS03;
	%QX3164.5 := AL_HI05_CONTROL_DEVIATION_DS04;
	%QX3164.6 := AL_HI05_CONTROL_DEVIATION_DS05;
	%QX3164.7 := AL_HI05_CONTROL_DEVIATION_DS07;
	%QX3167.0 := AL_HI05_CONTROL_DEVIATION_DS08;
	%QX3167.1 := AL_HI05_CONTROL_DEVIATION_DS09;
	%QX3167.2 := AL_HI05_CONTROL_DEVIATION_DS10;
	%QX3167.3 := AL_HI05_CONTROL_DEVIATION_DS11;
	%QX3167.4 := AL_HI05_CONTROL_DEVIATION_DS12;
	%QX3170.3 := AL_HI05_CONTROL_DEVIATION_DS14; // Verificar
	%QX3167.5 := AL_HI05_CONTROL_DEVIATION_DSTORRE;
END_IF

END_PROGRAM

// Device/Application/Transferencia
PROGRAM Transferencia
VAR
	//Tempos	
	
	//Tempo de estrela do mexedor principal
	TMR_ESTRELA_MH:TON;
	//Tempo retardo troca de estrela para triangulo mexedor principal
	TMR_RETARDO_TRIANGULO_MH:TON;
	
	
	//Boleanos
	
	//Libera triangulo moinho
	LIBERA_TRIANGULO_MH:BOOL;
	//Liga estrela moinho
	LIGA_ESTRELA_MH:BOOL;
	//Liga triangulo moinho
	LIGA_TRIANGULO_MH:BOOL;
	//Liga/desliga moinho
	LIGA_MOINHO:BOOL;
	//Transferencia em automatico
	TRANSFEREN_AUTO:BOOL;
	//Iniciou a transferencia
	INICIO_TRANSFERENCIA:BOOL;	
	//Bomba de transferencia desligada na espera
	BBTRANS_DESLIGADO_NA_ESPERA:BOOL;
	CONVERT_PRESSAO_VEL_BB: LIN_TRAFO;
	BLINK_BB: BLINK;
	ATUALIZA_VELOC_BB: BOOL;
	
END_VAR

// Lógica da transferencia da pasta do processo Slurry Making para o processo Spay Drying

//=================================================================================================
// Controle manual dos equipamentos 
//=================================================================================================

IF BTS_MASLU = FALSE THEN

	//Bomba Transferencia =======================================
	
	IF BTS_BBTRANSF = TRUE AND SD_VLMISTURA = TRUE AND  AL_GERAL = FALSE THEN
		IF SD_BBTRANS = TRUE THEN
			SD_BBTRANS := FALSE;
		ELSE
			SD_BBTRANS := TRUE;
		END_IF		
		BTS_BBTRANSF := FALSE;	
	ELSIF AL_GERAL = TRUE OR SD_VLMISTURA = FALSE THEN
		SD_BBTRANS := FALSE;
		BTS_BBTRANSF := FALSE;
	END_IF
		
	
	//Leitura de pressao maxima na linha de alta ======================
	
	IF LEITURA_PRES_LA > PRST_MAX_PRESSAO_BA THEN
		PRESSAO_ALTA_LINHA_ALTA := TRUE;
	ELSE
		PRESSAO_ALTA_LINHA_ALTA := FALSE;
	END_IF
	
		
	//Se alarme geral deliga tudo =======================================================
	
	IF AL_GERAL = TRUE THEN
		
		LIGA_MOINHO := FALSE;
		SD_BB := FALSE;
		SD_BA1 := FALSE;
		SD_BA2 := FALSE;
		SD_MXESPERA := FALSE;
		SD_BBTRANS := FALSE;
		INICIO_TRANSFERENCIA :=FALSE;
		
	END_IF
	
	//Memorias do automatico que devem ser desligadas
	TRANSFEREN_AUTO := FALSE;
ELSE
	// comando automatico ===================================================
	
	//transferencia em automatico
	IF AL_GERAL = FALSE THEN
		TRANSFEREN_AUTO := TRUE;
	ELSE
		TRANSFEREN_AUTO := FALSE;
	END_IF	
	
	//bomba de transferencia =================================
	//se auto + transferencia ativada + transferencia nunca iniciou + nivel maximo misturador de espera
	IF TRANSFEREN_AUTO = TRUE AND TRANSFERENCIA_lIBERADA = TRUE AND INICIO_TRANSFERENCIA = FALSE AND LEITURA_NI_MXESPE < PRST_MAX_MISTESPERA AND BBTRANS_DESLIGADO_NA_ESPERA = FALSE THEN
		INICIO_TRANSFERENCIA :=TRUE;
		SD_BBTRANS := TRUE;
	//se auto + transferencia ativada + transferencia ja iniciou uma vez + nivel reeligamento bomba transfe.
	ELSIF TRANSFEREN_AUTO = TRUE AND TRANSFERENCIA_lIBERADA = TRUE AND INICIO_TRANSFERENCIA = TRUE AND LEITURA_NI_MXESPE < PRST_TOL_NIVEL_MXESP_BT THEN
		SD_BBTRANS := TRUE;
		BBTRANS_DESLIGADO_NA_ESPERA := FALSE;
	ELSIF LEITURA_NI_MXESPE >= PRST_MAX_MISTESPERA AND LEITURA_NI_MXESPE > PRST_TOL_NIVEL_MXESP_BT THEN
		SD_BBTRANS := FALSE;
		BBTRANS_DESLIGADO_NA_ESPERA := TRUE;
	ELSIF TRANSFEREN_AUTO = FALSE OR TRANSFERENCIA_lIBERADA = FALSE THEN
		BBTRANS_DESLIGADO_NA_ESPERA := FALSE;
		SD_BBTRANS := FALSE;
	END_IF
		
END_IF


//=================================================================================================
// Controles que independem do manual/automatico 
//=================================================================================================

//Leitura de pressao maxima na linha de alta =============
	
	IF LEITURA_PRES_LA > PRST_MAX_PRESSAO_BA THEN
		PRESSAO_ALTA_LINHA_ALTA := TRUE;
	ELSE
		PRESSAO_ALTA_LINHA_ALTA := FALSE;
	END_IF

	//Mexedor de espera  =====================================
	
	IF BTS_MXE = TRUE AND AL_GERAL = FALSE  THEN
		IF SD_MXESPERA = TRUE THEN
			SD_MXESPERA := FALSE;
		ELSE
			SD_MXESPERA := TRUE;
		END_IF
		BTS_MXE := FALSE;
	ELSIF AL_GERAL = TRUE THEN
		SD_MXESPERA := FALSE;
		BTS_MXE := FALSE;
	END_IF
	

(*//Moinho  ================================================
	
	IF BTS_MH = TRUE AND AL_MHE = FALSE AND AL_GERAL = FALSE THEN
		IF LIGA_MOINHO = TRUE THEN
			LIGA_MOINHO := FALSE;
		ELSE
			LIGA_MOINHO := TRUE;
		END_IF		
		BTS_MH := FALSE;	
	ELSIF  AL_MHE = TRUE OR	AL_GERAL = TRUE  THEN
		LIGA_MOINHO := FALSE;
		BTS_MH := FALSE;
	END_IF
	
	//comando estrela
	//LIGA ESTRELA	
	IF LIGA_MOINHO = TRUE AND AL_MHE = FALSE  THEN
		IF LIGA_ESTRELA_MH = FALSE THEN
			SD_MH_E := TRUE;
		ELSE
			SD_MH_E := FALSE;
		END_IF
		LIBERA_TRIANGULO_MH := TRUE;
	ELSE
		SD_MH_E := FALSE;	
		LIBERA_TRIANGULO_MH:=FALSE;
	END_IF
	
	//TEMPO PARA ENTRAR O TRIANGULO
	TMR_ESTRELA_MH(IN:= LIBERA_TRIANGULO_MH, PT:= T#5S);	
	LIGA_ESTRELA_MH := TMR_ESTRELA_MH.Q;
	//TEMPO DE INTERVALO ENTRE ESTRELA E TRIANGULO
	TMR_RETARDO_TRIANGULO_MH(IN:= LIGA_ESTRELA_MH, PT:= T#0.2S);
	LIGA_TRIANGULO_MH := TMR_RETARDO_TRIANGULO_MH.Q;
	SD_MH_T := LIGA_TRIANGULO_MH;
	
	IF LIBERA_TRIANGULO_MH = TRUE THEN
		SD_MH_P := TRUE;
	ELSE
		SD_MH_P := FALSE;
	END_IF*)

//libera valvula de sopro =======================================================
IF BTS_HAB_SOPRO_SEMPH = TRUE THEN
	IF SOPRO_SEM_PH = TRUE THEN
		SOPRO_SEM_PH := FALSE;
	ELSE
		SOPRO_SEM_PH := TRUE;	
	END_IF
	BTS_HAB_SOPRO_SEMPH := FALSE;
END_IF

//Valvula de retorno =========================================================

//Libera sopro ====================================================================
IF SOPRO_SEM_PH = FALSE THEN
	IF AL_GERAL = FALSE AND (ED_PNM1_L = TRUE AND ED_PNM2_L = TRUE AND ED_PNM3_L = TRUE AND ED_PNM4_L = TRUE AND 
	ED_ESTSAIRLF_L = TRUE AND ED_ESTST_L = TRUE ) OR BTS_LIBERA_SEMPH = TRUE AND  PRESSAO_ALTA_LINHA_ALTA = FALSE THEN
		SOPRO_LIBERADO := TRUE;
	ELSIF PRESSAO_ALTA_LINHA_ALTA = TRUE THEN
		SOPRO_LIBERADO := FALSE;
	ELSE
		SOPRO_LIBERADO := FALSE;
	END_IF
ELSE
	SOPRO_LIBERADO := TRUE;
END_IF

			
//libera valvula de sopro
IF BTS_VLR = TRUE  THEN
	IF SD_VLR = TRUE THEN
		SD_VLR := FALSE;
	ELSE
		SD_VLR := TRUE;	
	END_IF
	    BTS_VLR := FALSE;
END_IF


//Bombas ==========================================================
	
//Bomba baixa ================================
		
IF BTS_BB = TRUE  AND NIVEL_MINIMO_MXE = FALSE AND AL_GERAL = FALSE AND PRESSAO_ALTA_LINHA_ALTA = FALSE AND BB_02_ST = FALSE THEN //INTERTRAVAMENTO COM A BOMBA 02 E 03 (AMPLIAÇÃO)
	IF SD_BB = TRUE THEN
		SD_BB := FALSE;
	ELSE
		SD_BB := TRUE;
	END_IF	
	BTS_BB := FALSE;
ELSIF  AL_GERAL = TRUE OR NIVEL_MINIMO_MXE = TRUE THEN
	SD_BB := FALSE;
	BTS_BB := FALSE;
END_IF
	

//move velocidade 

//IF SD_BB = TRUE  THEN
	//Vel_BB := PRST_VEL_BB;
	
	//PRESSAO_BOMBA :=PRST_PRESS_BB;
	//CONVERT_PRESSAO_VEL_BB(IN:=LEITURA_PRES_LB, IN_MIN:= (PRST_PRESS_BB*0.9), IN_MAX:=(PRST_PRESS_BB*1.1),OUT_MIN:=0, OUT_MAX:=100);
		//PRESSAO_BOMBA :=CONVERT_PRESSAO_VEL_BB.OUT;
//ELSE
	//Vel_BB:= 0;
//END_IF


//========================PRESSAO BOMBA DE BAIXA================
IF PRESSAO_BOMBA > 99 THEN
	PRESSAO_BOMBA := 100;
END_IF

IF PRESSAO_BOMBA < 1 THEN
	PRESSAO_BOMBA := 0;
END_IF


IF (SD_BB = TRUE AND BB_AUTOM = TRUE) AND LEITURA_PRES_LB <  (PRST_PRESS_BB*0.9)  THEN
		PRESSAO_BOMBA := PRESSAO_BOMBA+0.03;
		
		

END_IF

IF (SD_BB = TRUE AND BB_AUTOM = TRUE) AND LEITURA_PRES_LB <  (PRST_PRESS_BB*0.7)  THEN
		PRESSAO_BOMBA := PRESSAO_BOMBA+0.1;
		
		

END_IF

IF (SD_BB = TRUE AND BB_AUTOM = TRUE) AND (LEITURA_PRES_LB <  PRST_PRESS_BB*1.03 AND LEITURA_PRES_LB > PRST_PRESS_BB*0.97)  THEN
		PRESSAO_BOMBA := PRESSAO_BOMBA;
		
		END_IF

IF (SD_BB = TRUE AND BB_AUTOM = TRUE) AND (LEITURA_PRES_LB <  PRST_PRESS_BB AND LEITURA_PRES_LB >  PRST_PRESS_BB*0.9)  THEN
		PRESSAO_BOMBA := PRESSAO_BOMBA+0.001;
		END_IF
		
		IF (SD_BB = TRUE AND BB_AUTOM = TRUE) AND (LEITURA_PRES_LB > PRST_PRESS_BB AND LEITURA_PRES_LB <  PRST_PRESS_BB*1.1)  THEN
		PRESSAO_BOMBA := PRESSAO_BOMBA-0.001;
		
END_IF



IF (SD_BB = TRUE AND BB_AUTOM = TRUE) AND LEITURA_PRES_LB >  (PRST_PRESS_BB*1.1) THEN
	PRESSAO_BOMBA := PRESSAO_BOMBA-0.03;
	

END_IF


IF (SD_BB = TRUE AND BB_AUTOM = TRUE) AND LEITURA_PRES_LB >  (PRST_PRESS_BB*1.3) THEN
	PRESSAO_BOMBA := PRESSAO_BOMBA-0.1;
	

END_IF

IF BB_AUTOM = FALSE AND BTS_BB_AUTOM = TRUE THEN
	BB_AUTOM := TRUE;
	BTS_BB_AUTOM :=FALSE;
END_IF

IF BB_AUTOM = TRUE AND BTS_BB_AUTOM = TRUE THEN
	BB_AUTOM := FALSE;
	BTS_BB_AUTOM :=FALSE;
END_IF

//move velocidade em manual
IF (SD_BB = TRUE AND BB_AUTOM = FALSE) THEN
	Vel_BB := PRST_VEL_BB;
	PRESSAO_BOMBA := Vel_BB;
	END_IF


//move velocidade em automatico, buscando a pressão setada
//======================blink===========
//BLINK_BB(ENABLE:= TRUE, TIMELOW:= T#10S, TIMEHIGH:= T#0.1S, OUT=> ATUALIZA_VELOC_BB);
//IF ATUALIZA_VELOC_BB = TRUE THEN
	
	IF (SD_BB = TRUE AND BB_AUTOM = TRUE ) THEN
	Vel_BB := PRESSAO_BOMBA;
	END_IF

	
//END_IF
//====================blink===========


	IF SD_BB = FALSE THEN
	Vel_BB:= 0;
	END_IF
	

//========================PRESSAO BOMBA DE BAIXA================	
		
//Sempre quando trabalha com duas bombas liadas, suas velocidades são iguais, sendo assim vou pegar a alteração no PRST_VEL_BA1
//e espelhar para a BA2
//Bomba alta 1 ================================
	
IF BTS_BA1 = TRUE   AND SD_BB=TRUE AND AL_GERAL = FALSE AND  PRESSAO_ALTA_LINHA_ALTA = FALSE THEN
IF (NOT SD_BA2) OR (NOT BA_03_ST) THEN //INTERTRAVAMENTO COM A BOMBA 02 E 03 (AMPLIAÇÃO)
IF SD_BA1 = TRUE THEN
		SD_BA1 := FALSE;
	ELSE
		SD_BA1 := TRUE;
	END_IF
	BTS_BA1 := FALSE;
	END_IF
ELSIF AL_GERAL = TRUE OR SD_BB = FALSE THEN
	SD_BA1 := FALSE;
	BTS_BA1 := FALSE;

END_IF
	
//move velocidade
IF SD_BA1 = TRUE THEN
	VEL_ALT1 := PRST_VEL_BA1;
ELSE
	VEL_ALT1:= 0;
END_IF
		
//Sempre quando trabalha com duas bombas liadas, suas velocidades são iguais, sendo assim vou pegar a alteração no PRST_VEL_BA1
//e espelhar para a BA2
//Bomba alta 2 =================================
	
IF BTS_BA2 = TRUE  AND SD_BB=TRUE AND AL_GERAL = FALSE AND  PRESSAO_ALTA_LINHA_ALTA = FALSE THEN
IF (NOT SD_BA1) OR (NOT BA_03_ST) THEN	//INTERTRAVAMENTO COM A BOMBA 01 E 03 (AMPLIAÇÃO)
IF SD_BA2 = TRUE THEN
		SD_BA2 := FALSE;
	ELSE
		SD_BA2 := TRUE;
	END_IF
	BTS_BA2 := FALSE;
	END_IF
ELSIF AL_GERAL = TRUE OR SD_BB = FALSE  THEN
	SD_BA2 := FALSE;
	BTS_BA2 := FALSE;
END_IF	
	
//move velocidade
IF SD_BA2 = TRUE THEN			
	VEL_ALT2 := PRST_VEL_BA1;		
ELSE
	VEL_ALT2:= 0;
END_IF

			
//Bomba de lubrificacao da bomba de alta 1 =====================================

IF SD_BA1 = TRUE THEN
	SD_BLBA1 := TRUE;
ELSE
	SD_BLBA1 := FALSE;
END_IF


//Bomba de lubrificacao da bomba de alta 2 =====================================

IF SD_BA2 = TRUE THEN
	SD_BLBA2 := TRUE;
ELSE
	SD_BLBA2 := FALSE;
END_IF

END_PROGRAM

// Device/Application/Status
PROGRAM Status
VAR
	// Valvulas de descargas abertas
	DescargasAbertas: BOOL;
END_VAR

// POU de status dos equipamentos

// Carga de materiais =============================================================

//Rosca de Pó 1  Ligada
IF ED_RPO1_L OR SD_RPO1 THEN
	%QX3121.0:= TRUE;
ELSE
	%QX3121.0:= FALSE;
END_IF

//Rosca de Pó 2  Ligada
IF ED_RPO2_L OR SD_RPO2 THEN
	%QX3121.1:= TRUE;
ELSE
	%QX3121.1:= FALSE;
END_IF

//Rosca de Pó 3  Ligada
IF ED_RPO3_L OR SD_RPO3 THEN
	%QX3121.2:= TRUE;
ELSE
	%QX3121.2:= FALSE;
END_IF

//Rosca de Pó 4  Ligada
IF ED_RPO4_L  OR SD_RPO4 THEN
	%QX3121.3:= TRUE;
ELSE
	%QX3121.3:= FALSE;
END_IF

//Rosca de Pó 5  Ligada
IF ED_RPO5_L OR SD_RPO5 THEN
	%QX3121.4:= TRUE;
ELSE
	%QX3121.4:= FALSE;
END_IF

//Rosca 6 Horizontal
IF ED_RC6H_L  THEN
	%QX3121.5:= TRUE;
ELSE
	%QX3121.5:= FALSE;
END_IF

//Rosca 7 inclinada
IF ED_RC7I_L  THEN
	%QX3121.6:= TRUE;
ELSE
	%QX3121.6:= FALSE;
END_IF


//Balança de liquidos 1 carga rapida ligada
IF SD_BLL1R = TRUE THEN
	%QX3123.0:= TRUE;
ELSE
	%QX3123.0:= FALSE;
END_IF

//Balança de liquidos 1 carga lenta ligada
IF SD_BLL1L = TRUE  THEN
	%QX3123.1:= TRUE;
ELSE
	%QX3123.1:= FALSE;
END_IF


//Balança de liquidos 2 carga rapida ligada
IF SD_BLL2R = TRUE THEN
	%QX3123.2:= TRUE;
ELSE
	%QX3123.2:= FALSE;
END_IF

//Balança de liquidos 2 carga lenta ligada
IF SD_BLL2L = TRUE THEN
	%QX3123.3:= TRUE;
ELSE
	%QX3123.3:= FALSE;
END_IF


//Balança de liquidos 3 carga rapida ligada
IF SD_BLL3R = TRUE THEN
	%QX3123.4:= TRUE;
ELSE
	%QX3123.4:= FALSE;
END_IF

//Balança de liquidos 3 carga lenta ligada
IF SD_BLL3L = TRUE THEN
	%QX3123.5:= TRUE;
ELSE
	%QX3123.5:= FALSE;
END_IF


//Balança de liquidos 4 carga rapida ligada
IF SD_BLL4R = TRUE THEN
	%QX3123.6:= TRUE;
ELSE
	%QX3123.6:= FALSE;
END_IF

//Balança de liquidos 4 carga lenta ligada
IF SD_BLL4L = TRUE THEN
	%QX3123.7:= TRUE;
ELSE
	%QX3123.7:= FALSE;
END_IF

//Valvulas de descargas ===============================================================

//Balança de sólido 1 descarga ligada
IF ED_BLS1D_L = FALSE THEN
	%QX3121.7:= TRUE;
ELSE
	%QX3121.7:= FALSE;
END_IF

//Balança de sólido 2 descarga ligada
IF ED_BLS2D_L  = FALSE THEN
	%QX3120.0:= TRUE;
ELSE
	%QX3120.0:= FALSE;
END_IF

//Balança de sólido 3 descarga ligada
IF ED_BLS3D_L  = FALSE THEN
	%QX3120.1:= TRUE;
ELSE
	%QX3120.1:= FALSE;
END_IF

//Balança de sólido 4 descarga ligada
IF ED_BLS4D_L  = FALSE THEN
	%QX3120.2:= TRUE;
ELSE
	%QX3120.2:= FALSE;
END_IF

//Balança de sólido 5 descarga ligada
IF ED_BLS5D_L  = FALSE THEN
	%QX3120.3:= TRUE;
ELSE
	%QX3120.3:= FALSE;
END_IF

//Balança de liquidos 1 descarga ligada
IF SD_BLL1D  THEN
	%QX3120.4:= TRUE;
ELSE
	%QX3120.4:= FALSE;
END_IF

//Balança de liquidos 2 descarga ligada
IF SD_BLL2D  THEN
	%QX3120.5:= TRUE;
ELSE
	%QX3120.5:= FALSE;
END_IF

//Balança de liquidos 3 descarga ligada
IF SD_BLL3D  THEN
	%QX3120.6:= TRUE;
ELSE
	%QX3120.6:= FALSE;
END_IF

//Balança de liquidos 4 descarga ligada
IF SD_BLL4D  THEN
	%QX3120.7:= TRUE;
ELSE
	%QX3120.7:= FALSE;
END_IF


//Valvulas =====================================================================

//valvula saida mexedor aberta
IF SD_VLMISTURA THEN
	%QX3126.6 := TRUE;
ELSE
	%QX3126.6 := FALSE;
END_IF


//Valvula de vapor
IF SD_VPMECEDOR = TRUE THEN
	%QX3129.0 := TRUE;
ELSE
	%QX3129.0 := FALSE;
END_IF

// Mexedores ===================================================================

//Mexedor principal
IF ED_CFMXP_P = TRUE AND ED_CFMXP_T = TRUE THEN
	%QX3122.0 := TRUE;
	ST_CFMXP := TRUE;
ELSE
	%QX3122.0 := FALSE;
	ST_CFMXP := FALSE;
END_IF



//Mexedor de espera
IF SD_MXESPERA = TRUE THEN
	%QX3122.1 := TRUE;
ELSE
	%QX3122.1 := FALSE;
END_IF



// Bombas ===============================================================================

//Boma de combustivel
IF ED_BOCOMB_L = TRUE THEN
	%QX3122.2 := TRUE;
ELSE
	%QX3122.2 := FALSE;
END_IF

//Boma Diesel para piloto
IF ED_BDP_L = TRUE THEN
	%QX3122.3 := TRUE;
ELSE
	%QX3122.3 := FALSE;
END_IF

//Boma de Baixa
IF SD_BB = TRUE THEN
	%QX3122.4 := TRUE;
ELSE
	%QX3122.4 := FALSE;
END_IF

//Boma de Alta 1
IF SD_BA1 = TRUE THEN
	%QX3122.5 := TRUE;
ELSE
	%QX3122.5 := FALSE;
END_IF

//Boma de Alta 2
IF SD_BA2 = TRUE THEN
	%QX3122.6 := TRUE;
ELSE
	%QX3122.6 := FALSE;
END_IF

//Boma de Transferencia
IF SD_BBTRANS = TRUE AND ED_BTRA_D = TRUE THEN
	%QX3124.4 := TRUE;
ELSE
	%QX3124.4 := FALSE;
END_IF

//Bomba acusol
IF SD_BACU = TRUE THEN
	%QX3129.5 := TRUE;
ELSE
	%QX3129.5 := FALSE;
END_IF

//Bomba blend
IF SD_BBD = TRUE THEN
	%QX3128.4 := TRUE;
ELSE
	%QX3128.4 := FALSE;
END_IF

//Bomba silicato
IF SD_BSIL = TRUE THEN
	%QX3128.5 := TRUE;
ELSE
	%QX3128.5 := FALSE;
END_IF

//Bomba Sulfonico
IF SD_BSUL = TRUE THEN
	%QX3128.6 := TRUE;
ELSE
	%QX3128.6 := FALSE;
END_IF

//Bomba Soda
IF SD_BSOD = TRUE THEN
	%QX3128.7 := TRUE;
ELSE
	%QX3128.7 := FALSE;
END_IF
	
//Bomba Soda
IF SD_BAG = TRUE THEN
	%QX3131.0 := TRUE;
ELSE
	%QX3131.0 := FALSE;
END_IF		
		
//Bomba Perfume 1
IF SD_BPER1 = TRUE THEN
	%QX3131.1 := TRUE;
ELSE
	%QX3131.1 := FALSE;
END_IF	

//Bomba Perfume 2
IF SD_BPER2 = TRUE THEN
	%QX3131.2 := TRUE;
ELSE
	%QX3131.2 := FALSE;
END_IF	

(*//Moinho =============================================================
IF ED_CFMH_P = TRUE AND ED_CFMH_T = TRUE THEN
	%QX3125.0 := TRUE;
ELSE
	%QX3125.0 := FALSE;
END_IF*)

//Exaustores ==========================================================

//FM1
IF ED_CFEXFM1_P = TRUE AND ED_CFEXFM1_T = TRUE THEN
	%QX3125.1 := TRUE;
ELSE
	%QX3125.1 := FALSE;
END_IF

//FM2
IF ED_CFEXFM2_P = TRUE AND ED_CFEXFM2_T = TRUE THEN
	%QX3125.2 := TRUE;
ELSE
	%QX3125.2 := FALSE;
END_IF

//Exaustor da torre
IF SD_EX125 = TRUE AND  AL_EXTORRE = FALSE THEN
	%QX3124.7 := TRUE;
ELSE
	%QX3124.7 := FALSE;
END_IF

//Ventiladores ===========================================================

//Ventilador FM1
IF ED_CFVEXFM2_P = TRUE AND  ED_CFVEXFM2_T = TRUE THEN
	%QX3126.5 := TRUE;
ELSE
	%QX3126.5 := FALSE;
END_IF

//ventilador FM2
IF SD_VFLU = TRUE THEN
	%QX3129.3 := TRUE;
ELSE
	%QX3129.3 := FALSE;
END_IF

//ventilador Queimador 100CV
IF SD_EX100 = TRUE THEN
	%QX3126.7 := TRUE;
ELSE
	%QX3126.7 := FALSE;
END_IF

//Esteiras ===============================================================

//TC3
IF ED_TC3_L = TRUE  THEN
	%QX3125.4 := TRUE;
ELSE
	%QX3125.4 := FALSE;
END_IF

//Saida da torre
IF ED_ESTST_L = TRUE THEN
	%QX3129.1 := TRUE;
ELSE
	%QX3129.1 := FALSE;
END_IF

//TC02
IF SD_ESTTC02 = TRUE THEN
	%QX3129.4 := TRUE;
ELSE
	%QX3129.4 := FALSE;
END_IF

//TC09
IF SD_ESTTC9 = TRUE THEN
	%QX3131.6 := TRUE;
ELSE
	%QX3131.6 := FALSE;
END_IF

//TC10
IF SD_ESTTC10 = TRUE THEN
	%QX3131.7 := TRUE;
ELSE
	%QX3131.7 := FALSE;
END_IF

//TC13
IF SD_ESTTC13 = TRUE THEN
	%QX3130.0 := TRUE;
ELSE
	%QX3130.0 := FALSE;
END_IF

//TC12
IF SD_ESTTC12 = TRUE THEN
	%QX3130.1 := TRUE;
ELSE
	%QX3130.1 := FALSE;
END_IF

//TC08
IF SD_ESTTC8 = TRUE OR SD_ESTTC8_R = TRUE THEN
	%QX3130.2 := TRUE;
ELSE
	%QX3130.2 := FALSE;
END_IF

//TC08 Reversao
IF SD_ESTTC8_R = TRUE THEN
	%QX3130.3 := TRUE;
ELSE
	%QX3130.3 := FALSE;
END_IF

//Air Lifit ===============================================================

//Esteira saida do air lifit
IF ED_ESTSAIRLF_L = TRUE THEN
	%QX3125.5 := TRUE;
ELSE
	%QX3125.5 := FALSE;
END_IF

//Motor Air Lifit
IF SD_MAIRLIF = TRUE THEN
	%QX3125.6 := TRUE;
ELSE
	%QX3125.6 := FALSE;	
END_IF


//Elevadores =============================================================

//elevador 2
IF SD_EL2DMIX = TRUE THEN		
	%QX3125.7 := TRUE;
ELSE	
	%QX3125.7 := FALSE; 
END_IF

//elevador 4
IF SD_EL2 = TRUE THEN
	%QX3129.2 := TRUE;
ELSE
	%QX3129.2 := FALSE; 
END_IF

//Valvulas ================================================================

//Valvula retorno aberta
IF SD_VLR = FALSE THEN
	%QX3124.0 := TRUE;
ELSE
	%QX3124.0 := FALSE;
END_IF

//valvula retorno fechada
IF SD_VLR = TRUE THEN
	%QX3124.1 := TRUE;
ELSE
	%QX3124.1 := FALSE;
END_IF

//Queimador ===============================================================

IF SD_LQUEI = TRUE THEN
	%QX3122.7 := TRUE;
ELSE
	%QX3122.7 := FALSE;
END_IF



//Satus ligado Dosadores Schenck =======================================================

//DS1 - PB01
IF LIGA_DS1 = TRUE THEN
	%QX3127.0 := TRUE;
ELSE
	%QX3127.0 := FALSE;
END_IF

//DS11 - PB11
IF LIGA_DS11 = TRUE THEN
	%QX3127.1 := TRUE;
ELSE
	%QX3127.1 := FALSE;
END_IF

//DS2 
IF LIGA_DS2 = TRUE THEN
	%QX3127.2 := TRUE;
ELSE
	%QX3127.2 := FALSE;
END_IF

//DS3 
IF LIGA_DS3 = TRUE THEN
	%QX3127.3 := TRUE;
ELSE
	%QX3127.3 := FALSE;
END_IF

//DS4 
IF LIGA_DS4 = TRUE THEN
	%QX3127.4 := TRUE;
ELSE
	%QX3127.4 := FALSE;
END_IF

//DS5
IF LIGA_DS5 = TRUE THEN
	%QX3127.5 := TRUE;
ELSE
	%QX3127.5 := FALSE;
END_IF

//DS7 
IF DS07_HAB = TRUE THEN
	%QX3127.7 := TRUE;
ELSE
	%QX3127.7 := FALSE;
END_IF

//DS8
IF LIGA_DS8 = TRUE THEN
	%QX3126.0 := TRUE;
ELSE
	%QX3126.0 := FALSE;
END_IF

//DS9
IF LIGA_DS9 = TRUE THEN
	%QX3126.1 := TRUE;
ELSE
	%QX3126.1 := FALSE;
END_IF

//DS10
IF LIGA_DS10 = TRUE THEN
	%QX3126.2 := TRUE;
ELSE
	%QX3126.2 := FALSE;
END_IF

//DS12
IF LIGA_DS12 = TRUE THEN
	%QX3126.3 := TRUE;
ELSE
	%QX3126.3 := FALSE;
END_IF

//DS TORRE
IF DSATORRE_HAB = TRUE THEN
	%QX3126.4 := TRUE;
ELSE
	%QX3126.4 := FALSE;
END_IF

//DS14
IF LIGA_DS14 = TRUE THEN
	%QX3126.8 := TRUE;
ELSE
	%QX3126.8 := FALSE;
END_IF
//Dumper da torre ===================================================

//dumper para atm	
IF 	ED_DUPATM_A = TRUE AND ED_DUPTORRE_A = FALSE  THEN
	%QX3129.6 := TRUE;
ELSE
	%QX3129.6 := FALSE;
END_IF

//dumper para torre	
IF 	ED_DUPTORRE_A = TRUE AND ED_DUPATM_A = FALSE THEN
	%QX3129.7 := TRUE;
ELSE
	%QX3129.7 := FALSE;
END_IF

// Status do Soporo  Sem PH ==================================================
IF SOPRO_SEM_PH = TRUE THEN
	%QX3128.0 := TRUE;
ELSE
	%QX3128.0 := FALSE;
END_IF

//Slurry Making em automatico ========================================
IF BTS_MASLU = TRUE THEN
	%QX3128.2 := TRUE;
ELSE
	%QX3128.2 := FALSE;
END_IF

//Filtros de manga ===================================================

//1
IF LIGA_FTM1 = TRUE THEN
	%QX3131.3 := TRUE;
ELSE
	%QX3131.3 := FALSE;
END_IF

//2
IF LIGA_FTM2 = TRUE THEN
	%QX3131.4 := TRUE;
ELSE
	%QX3131.4 := FALSE;
END_IF

//Peneira ============================================================

IF SD_M1PN = TRUE THEN
	%QX3131.5 := TRUE;
ELSE
	%QX3131.5 := FALSE;
END_IF

//Status Gravimetrico Dosadoras Schenck ========================================

//DS1
IF %IX15031.3 = FALSE THEN
	%QX3133.0 := TRUE;
ELSE
	%QX3133.0 := FALSE;
END_IF

//DS2
IF %IX15033.3 = FALSE THEN
	%QX3133.1 := TRUE;
ELSE
	%QX3133.1 := FALSE;
END_IF

//DS3
IF %IX15035.3 = FALSE THEN
	%QX3133.2 := TRUE;
ELSE
	%QX3133.2 := FALSE;
END_IF

//DS4
IF %IX15037.3 = FALSE THEN
	%QX3133.3 := TRUE;
ELSE
	%QX3133.3 := FALSE;
END_IF


//DS5
IF %IX15039.3 = FALSE THEN
	%QX3133.4 := TRUE;
ELSE
	%QX3133.4 := FALSE;
END_IF

//DS7
IF %IX15041.3 = FALSE THEN
	%QX3133.5 := TRUE;
ELSE
	%QX3133.5 := FALSE;
END_IF


//DS8
IF %IX15043.3 = FALSE THEN
	%QX3133.6 := TRUE;
ELSE
	%QX3133.6 := FALSE;
END_IF

//DS9
IF %IX15045.3 = FALSE THEN
	%QX3133.7 := TRUE;
ELSE
	%QX3133.7 := FALSE;
END_IF

//DS10
IF %IX15047.3 = FALSE THEN
	%QX3132.0 := TRUE;
ELSE
	%QX3132.0 := FALSE;
END_IF

//DS11
IF %IX15049.3 = FALSE THEN
	%QX3132.1 := TRUE;
ELSE
	%QX3132.1 := FALSE;
END_IF

//DS12
IF %IX15051.3 = FALSE THEN
	%QX3132.2 := TRUE;
ELSE
	%QX3132.2 := FALSE;
END_IF

//DSTORRE
IF %IX15053.3 = FALSE THEN
	%QX3132.3 := TRUE;
ELSE
	%QX3132.3 := FALSE;
END_IF


//DS14
IF %IX15055.3 = FALSE THEN
	%QX3132.4 := TRUE;
ELSE
	%QX3132.4 := FALSE;
END_IF

// Ultima Carga ================================================================

IF ULTIMA_CARGA = TRUE THEN
	%QX3130.4 := TRUE;
ELSE
	%QX3130.4 := FALSE;
END_IF 

//PH em Automatico =============================================================
//PH1
IF BTS_MAPH1 = TRUE THEN
	%QX3130.5 := TRUE;
ELSE
	%QX3130.5 := FALSE;
END_IF

//PH2
IF BTS_MAPH2 = TRUE THEN
	%QX3130.6 := TRUE;
ELSE
	%QX3130.6 := FALSE;
END_IF

END_PROGRAM

// Device/Application/SprayDrying
PROGRAM SprayDrying
VAR
	//Informa dumper ligado
	DUMPER_LIGADO:BOOL;
	//Libera partida do Air Lift
	LIBERA_AIRLIFT:BOOL;
	
	//Libera tempo de aquisição
	LIBERA_TEMPO_AQUISICAO:BOOL;
	//Tempo de aquisição dos dados analógicos
	TEMPO_AQUISICAO:TON;
END_VAR

//     Processo Spray Drying - lógica do controle da fornalha e torre de secagem

//============================================================================
// comando que independe com controle manual/auto
//============================================================================

//Exaustor da torre (125 cv)==================================================
//Velocidade  de 0-100%
IF BTS_EXTORRE = TRUE  AND AL_GERAL = FALSE THEN	
	IF SD_EX125 = TRUE THEN
		SD_EX125 := FALSE;			
	ELSE
		SD_EX125 := TRUE;				
	END_IF		
	BTS_EXTORRE := FALSE;	
END_IF
//Deliga em caso de alarme
IF AL_GERAL = TRUE THEN
	SD_EX125 := FALSE;
	BTS_EXTORRE := FALSE;
END_IF
//move velocidade
IF SD_EX125 = TRUE THEN
	Vel_EXTORRE := PRST_VEL_EXTORRE;
ELSE
	Vel_EXTORRE := 0;
END_IF
		

//controle do Dumper Torre ===================================================
//se desligado, dumper para atmosfera, 
//se ligado, dumper para torre

IF BTS_DUMPER_TORRE = TRUE AND AL_GERAL = FALSE THEN	
	IF DUMPER_LIGADO = TRUE THEN
		DUMPER_LIGADO := FALSE;				
	ELSE
		DUMPER_LIGADO := TRUE;				
	END_IF
	BTS_DUMPER_TORRE := FALSE;
ELSIF AL_GERAL = TRUE THEN
	BTS_DUMPER_TORRE := FALSE;
	DUMPER_LIGADO := FALSE;
END_IF

//se a temperatura subir, joga dumper para atm
IF  TEMP_TORRE < PRST_SEGURANCA_TORRE AND DUMPER_LIGADO = TRUE THEN
	LIB_DUMPER := TRUE;
ELSE
	LIB_DUMPER := FALSE;
END_IF

//dumper para torre, primeiro abre para torre, depois fecha para atm
IF LIB_DUMPER = TRUE THEN
	SD_DUPTORRE := TRUE;	
	IF 	ED_DUPTORRE_A = TRUE AND ED_DUPTORRE_F = FALSE  THEN
		SD_DUPATM := FALSE;
	END_IF
END_IF
//dumper para atm, primeiro abre para atm, depois fecha para torre
IF LIB_DUMPER = FALSE THEN
	SD_DUPATM := TRUE;
	IF ED_DUPATM_A = TRUE AND ED_DUPATM_F = FALSE THEN
		SD_DUPTORRE := FALSE;
	END_IF
END_IF

//FECHA VÁLVULA DE RETORNO E ABRE O DUMPER PARA ATMOSFERA
IF  (AL_HI05_CONTROL_DEVIATION_DSTORRE = TRUE OR AL_HI05_CONTROL_DEVIATION_DS07 = TRUE OR PRESSAO_ALTA_LINHA_ALTA = TRUE)  THEN
	SD_DUPATM := TRUE;
	SD_VLR := FALSE;
	IF DUMPER_LIGADO = TRUE THEN
		DUMPER_LIGADO := FALSE;	
	END_IF	
	
	IF ED_DUPATM_A = TRUE AND ED_DUPATM_F = FALSE THEN
		SD_DUPTORRE := FALSE;
	END_IF
	
	
END_IF


//FECHA VÁLVULA DE RETORNO E ABRE O DUMPER PARA ATMOSFERA
//Ventilador do queimador (100 cv)==================================================

//Velocidade  de 0-100%
IF BTS_VENTIQUEIMADOR = TRUE  AND AL_GERAL = FALSE THEN	
	IF SD_EX100 = TRUE THEN
		SD_EX100 := FALSE;				
	ELSE
		SD_EX100 := TRUE;				
	END_IF
	BTS_VENTIQUEIMADOR := FALSE;
ELSIF AL_GERAL = TRUE THEN
	BTS_VENTIQUEIMADOR := FALSE;
	SD_EX100 := FALSE;
END_IF
//Deliga em caso de alarme
IF AL_GERAL = TRUE THEN
	SD_EX100 := FALSE;
	BTS_VENTIQUEIMADOR := FALSE;
END_IF
//move velocidade
IF SD_EX100 = TRUE AND ED_MAXVL100 = FALSE AND ED_MINVL100 = FALSE THEN
	VEL_VENTQUEIMADOR := PRST_VEL_VENTIQUEIMADOR;	
END_IF	
//comando para velocidade minima
IF SD_EX100 = TRUE AND ED_MINVL100 = TRUE THEN
	VEL_VENTQUEIMADOR := 55;
END_IF
//comando para velocidade maxima
IF SD_EX100 = TRUE AND ED_MAXVL100 = TRUE THEN
	VEL_VENTQUEIMADOR := 100;
END_IF
//se ventilador desligado zera saida analogica
IF  SD_EX100 = FALSE THEN
	VEL_VENTQUEIMADOR := 0;
END_IF


// Queimador =======================================================================

IF BTS_PARTIDAQUEIMADOR_REM = TRUE AND AL_GERAL = FALSE AND SD_EX100 = TRUE THEN
	IF SD_LQUEI = TRUE THEN
		SD_LQUEI := FALSE;
	ELSE
		SD_LQUEI := TRUE;
	END_IF
	BTS_PARTIDAQUEIMADOR_REM := FALSE;
ELSIF AL_GERAL = TRUE THEN
	BTS_PARTIDAQUEIMADOR_REM := FALSE;
	SD_LQUEI := FALSE;
END_IF


//Air Lift ====================================================================

IF BTS_VELAIRLF = TRUE AND AL_GERAL = FALSE AND ED_VELAIRLF100 = FALSE  THEN
	IF LIBERA_AIRLIFT = TRUE  THEN
		LIBERA_AIRLIFT := FALSE;
	ELSE
		LIBERA_AIRLIFT := TRUE;
	END_IF
	BTS_VELAIRLF := FALSE;	
ELSIF AL_GERAL = TRUE THEN
	BTS_VELAIRLF := FALSE;
	LIBERA_AIRLIFT := FALSE;
END_IF 

//libera motor
IF LIBERA_AIRLIFT = TRUE  THEN	
	SD_MAIRLIF:= TRUE;
ELSE	
	SD_MAIRLIF:= FALSE;
END_IF 

//Esteira saida Air Lift ======================================================

IF SD_ESTSTORRE = TRUE THEN	
	SD_ESTSAIRLIF:= TRUE;
ELSE
	SD_ESTSAIRLIF:= FALSE;	
END_IF 


//Esteira saida torre ==========================================================

IF BTS_ESTSATORRE = TRUE AND AL_GERAL = FALSE AND SOPRO_SEM_PH = FALSE THEN
	IF SD_ESTSTORRE = TRUE THEN
		SD_ESTSTORRE:= FALSE;
	ELSE
		SD_ESTSTORRE:= TRUE;	
	END_IF 
	BTS_ESTSATORRE := FALSE;
ELSIF BTS_ESTSATORRE = TRUE AND AL_GERAL = FALSE AND SOPRO_SEM_PH = TRUE THEN
	IF SD_ESTSTORRE = TRUE THEN
		SD_ESTSTORRE:= FALSE;
	ELSE
		SD_ESTSTORRE:= TRUE;	
	END_IF 
	BTS_ESTSATORRE := FALSE;
ELSIF AL_GERAL = TRUE THEN
	SD_ESTSTORRE:= FALSE;
	BTS_ESTSATORRE := FALSE;
END_IF 


//Esteira TC02 =================================================================
IF BTS_ESTTC02 = TRUE AND AL_GERAL = FALSE AND SOPRO_SEM_PH = FALSE THEN
	IF SD_ESTTC02 = TRUE THEN
		SD_ESTTC02:= FALSE;
	ELSE
		SD_ESTTC02:= TRUE;	
	END_IF 
	BTS_ESTTC02 := FALSE;
ELSIF BTS_ESTTC02 = TRUE AND AL_GERAL = FALSE AND SOPRO_SEM_PH = TRUE THEN
	IF SD_ESTTC02 = TRUE THEN
		SD_ESTTC02:= FALSE;
	ELSE
		SD_ESTTC02:= TRUE;	
	END_IF 
	BTS_ESTTC02 := FALSE;
ELSIF AL_GERAL = TRUE THEN
	SD_ESTTC02:= FALSE;
	BTS_ESTTC02 := FALSE;
END_IF 


//Esteira saida dosador Sulfato da Torre ==================================================

IF LIGA_DSTORRE = TRUE AND  AL_GERAL=FALSE  THEN	
	SD_ESTDSSUL := TRUE;
ELSE
	SD_ESTDSSUL := FALSE;
END_IF


// Libera aquisição de dados de pressões e temperatura ====================================

//Reseta o status de realizar aquisicao no supervisório
IF PRST_RESET_LEITURA_ANALOICA = 1 THEN
	GRAVAR_DADOS_ANALOGICAS := 0;
	PRST_RESET_LEITURA_ANALOICA := 0;
END_IF

//Libera contagem do tempo
IF SD_EX100 = TRUE AND TEMPO_AQUISICAO.Q = FALSE THEN	
	LIBERA_TEMPO_AQUISICAO := TRUE;
ELSE
	LIBERA_TEMPO_AQUISICAO := FALSE;
END_IF
	
TEMPO_AQUISICAO(IN:=LIBERA_TEMPO_AQUISICAO, PT:= T#1800S);

IF TEMPO_AQUISICAO.Q = TRUE THEN
	GRAVAR_DADOS_ANALOGICAS := 1;
END_IF

//===============Cálcula quantidade de Jatos abertos para exibir no relatório=============

IF SD_VLR = FALSE THEN
	QTD_JATOS :=0;
END_IF

IF LEITURA_BASE_SOP_TORRE >200 AND LEITURA_BASE_SOP_TORRE <1500 AND  SD_VLR = TRUE THEN
	QTD_JATOS :=1;
	
END_IF

IF LEITURA_BASE_SOP_TORRE >1500 AND LEITURA_BASE_SOP_TORRE <2500  AND SD_VLR = TRUE THEN
	QTD_JATOS :=2;
	
END_IF

	IF LEITURA_BASE_SOP_TORRE >2500 AND LEITURA_BASE_SOP_TORRE <3500 AND SD_VLR = TRUE THEN
	QTD_JATOS :=3;
	END_IF
	
	IF LEITURA_BASE_SOP_TORRE >3500 AND LEITURA_BASE_SOP_TORRE <4500 AND SD_VLR = TRUE THEN
	QTD_JATOS :=4;
	
END_IF

	IF LEITURA_BASE_SOP_TORRE >4500 AND LEITURA_BASE_SOP_TORRE <5500 AND SD_VLR = TRUE THEN
	QTD_JATOS :=5;
	
END_IF

	IF LEITURA_BASE_SOP_TORRE >5500 AND LEITURA_BASE_SOP_TORRE <6500 AND SD_VLR = TRUE THEN
	QTD_JATOS :=6;
	
END_IF

IF LEITURA_BASE_SOP_TORRE >6500 AND LEITURA_BASE_SOP_TORRE <7500 AND SD_VLR = TRUE THEN
	QTD_JATOS :=7;
	
END_IF

IF LEITURA_BASE_SOP_TORRE >7500 AND LEITURA_BASE_SOP_TORRE <8500 AND SD_VLR = TRUE THEN
	QTD_JATOS :=8;
	
END_IF
IF LEITURA_BASE_SOP_TORRE >8500 AND LEITURA_BASE_SOP_TORRE <9500 AND SD_VLR = TRUE THEN
	QTD_JATOS :=9;
	
END_IF
IF LEITURA_BASE_SOP_TORRE >9500 AND LEITURA_BASE_SOP_TORRE <10500 AND SD_VLR = TRUE THEN
	QTD_JATOS :=10;
	
END_IF

IF LEITURA_BASE_SOP_TORRE >10500 AND LEITURA_BASE_SOP_TORRE <11500 AND SD_VLR = TRUE THEN
	QTD_JATOS :=11;
	
END_IF

IF LEITURA_BASE_SOP_TORRE >11500 AND LEITURA_BASE_SOP_TORRE <12500 AND SD_VLR = TRUE THEN
	QTD_JATOS :=12;
	
END_IF
//===============Cálcula quantidade de Jatos abertos para exibir no relatório=============

END_PROGRAM

// Device/Application/AutoPH
PROGRAM AutoPH
VAR
		//Controle PH1
	CONTROLEPH1:LIN_TRAFO;
	//Velocidade automatica do PH1
	VELOCIDADEPH1AUTO:REAL;
	//preset de producao em KG do PH1 DE
	PRST_PRODUCAO_DE_PH1_KG:REAL;
	//preset de producao em KG do PH1 A
	PRST_PRODUCAO_A_PH1_KG:REAL;
	//Espera o fluidizador baixar para o peso minino, pois atingiu o peso maximo Ph1
	ESPERA_FLUIDIZADOR_BAIXAR_PESO_PH1:BOOL;
	
	
	//Controle PH2
	controlePH2:LIN_TRAFO;	
	//Velocidade automatica do PH2
	velocidadePH2Auto:REAL;
	//preset de producao em KG do PH2 DE
	PRST_PRODUCAO_DE_PH2_KG:REAL;
	//preset de producao em KG do PH2 A
	PRST_PRODUCAO_A_PH2_KG:REAL;
	//Espera o fluidizador baixar para o peso minino, pois atingiu o peso maximo Ph1
	ESPERA_FLUIDIZADOR_BAIXAR_PESO_PH2:BOOL;
		

END_VAR

// Controle automatico do PH1 ============================================================

//Conversão de Toneladas enviado pelo supervisório para Kg
PRST_PRODUCAO_A_PH1_KG := PRST_PRODUCAO_PH1_A * 1000;
PRST_PRODUCAO_DE_PH1_KG:= PRST_PRODUCAO_PH1_DE * 1000;

//Função de controle
CONTROLEPH1(IN:=LEITURA_PESO_FLUI1 , IN_MIN:=PRST_PESO_MIN_FLUID1, IN_MAX:=PRST_PESO_MAX_FLUID1,OUT_MIN:=PRST_PRODUCAO_A_PH1_KG, OUT_MAX:=PRST_PRODUCAO_DE_PH1_KG);
VELOCIDADEPH1AUTO:= CONTROLEPH1.OUT;

//verifica limites de peso maximo e minimo
//zera velocidade do ph com peso maximo
IF LEITURA_PESO_FLUI1 >= PRST_PESO_MAX_FLUID1 THEN
	ESPERA_FLUIDIZADOR_BAIXAR_PESO_PH1 := FALSE;
END_IF
	
//ativa velocidade do ph com peso minimo
IF LEITURA_PESO_FLUI1 <= PRST_PESO_MIN_FLUID1 THEN
	VELOCIDADEPH1AUTO:= PRST_PRODUCAO_A_PH1_KG;
	ESPERA_FLUIDIZADOR_BAIXAR_PESO_PH1 := FALSE;
END_IF
	
	
IF ESPERA_FLUIDIZADOR_BAIXAR_PESO_PH1 = FALSE AND BTS_MAPH1 = TRUE THEN
	//saida de controle ===============
	VELOCIDADE_PH1_AUTO := VELOCIDADEPH1AUTO;
ELSE
	VELOCIDADE_PH1_AUTO := 0;
END_IF

// Controle automatico do PH2 ============================================================

//Conversão de Toneladas enviado pelo supervisório para Kg
PRST_PRODUCAO_DE_PH2_KG := PRST_PRODUCAO_PH2_DE * 1000;
PRST_PRODUCAO_A_PH2_KG:= PRST_PRODUCAO_PH2_A * 1000;

//Função de controle
CONTROLEPH2(IN:=LEITURA_PESO_FLUI2 , IN_MIN:=PRST_PESO_MIN_FLUID2, IN_MAX:=PRST_PESO_MAX_FLUID2,OUT_MIN:=PRST_PRODUCAO_A_PH2_KG, OUT_MAX:=PRST_PRODUCAO_DE_PH2_KG);
VELOCIDADEPH2AUTO:= CONTROLEPH2.OUT;

//verifica limites de peso maximo e minimo
//zera velocidade do ph com peso maximo
IF LEITURA_PESO_FLUI2 >= PRST_PESO_MAX_FLUID2 THEN
	ESPERA_FLUIDIZADOR_BAIXAR_PESO_PH2 := FALSE;
END_IF
	
//ativa velocidade do ph com peso minimo
IF LEITURA_PESO_FLUI2 <= PRST_PESO_MIN_FLUID2 THEN
	VELOCIDADEPH2AUTO:= PRST_PRODUCAO_A_PH2_KG;
	ESPERA_FLUIDIZADOR_BAIXAR_PESO_PH2 := FALSE;
END_IF
	
	
IF ESPERA_FLUIDIZADOR_BAIXAR_PESO_PH2 = FALSE AND BTS_MAPH2 = TRUE THEN
	//saida de controle ===============
	VELOCIDADE_PH2_AUTO := VELOCIDADEPH2AUTO;
ELSE
	VELOCIDADE_PH2_AUTO := 0;
END_IF

END_PROGRAM

// Device/Application/FiltrosDeManga
PROGRAM FiltrosDeManga
VAR
	
	//Filtro de manga 1
	FTM1_TEMPO_BATIDA:TON;
	FTM1_TEMPO_INTERVALO_BATIDA:TON;	
	FTM1_LIBERA_BATIDA:BOOL;
	FTM1_LIBERA_INTERVALO_BATIDA:BOOL;
	FTM1_CONTADOR_CICLO_BATIDA:INT;
	FTM1_TEMPO_INTERVALO_BATIDA_TERMINOU:BOOL;	
	
	//Filtro de manga 2
	FTM2_TEMPO_BATIDA:TON;
	FTM2_TEMPO_INTERVALO_BATIDA:TON;	
	FTM2_LIBERA_BATIDA:BOOL;
	FTM2_LIBERA_INTERVALO_BATIDA:BOOL;
	FTM2_CONTADOR_CICLO_BATIDA:INT;
	FTM2_TEMPO_INTERVALO_BATIDA_TERMINOU:BOOL;	
END_VAR

//Filtro de manga 1 ==================================================================
	IF BTS_FILTM1 = TRUE  AND AL_GERAL = FALSE   THEN
		IF LIGA_FTM1 = TRUE THEN
			LIGA_FTM1 := FALSE;
		ELSE
			LIGA_FTM1 := TRUE;
		END_IF
		BTS_FILTM1 := FALSE;
	ELSIF AL_GERAL = TRUE THEN  //delsiga em caso de alarme
		LIGA_FTM1 := FALSE;
		BTS_FILTM1 := FALSE;
	END_IF

//ciclo de batidas
IF LIGA_FTM1 THEN
		
	//condição para iniciar primeiro ciclo
	IF NOT FTM1_LIBERA_INTERVALO_BATIDA  AND NOT FTM1_LIBERA_BATIDA THEN	
		FTM1_LIBERA_BATIDA:=TRUE;
	END_IF
	
	//tempo de pulso da batida
	FTM1_TEMPO_BATIDA(IN:=FTM1_LIBERA_BATIDA, PT:= T#1S);
	
	//ao final do tempo vai para o intervalo e incrementa o contador de filtro
	IF FTM1_TEMPO_BATIDA.Q THEN
		FTM1_CONTADOR_CICLO_BATIDA := FTM1_CONTADOR_CICLO_BATIDA + 1;
		FTM1_LIBERA_INTERVALO_BATIDA := TRUE;
		FTM1_LIBERA_BATIDA:=FALSE;
	END_IF
	
	//tempo de intervalo para cada batida
	FTM1_TEMPO_INTERVALO_BATIDA(IN:=FTM1_LIBERA_INTERVALO_BATIDA, PT:= T#30S);
	
	//ao final tempo de intervalo, faz a batida
	IF FTM1_TEMPO_INTERVALO_BATIDA.Q  THEN
		FTM1_LIBERA_BATIDA:=TRUE;
		FTM1_LIBERA_INTERVALO_BATIDA:= FALSE;
	END_IF	
	
	//se chegou no filtro 4, reinicia o ciclo dos filtros 1 - 4
	IF FTM1_LIBERA_INTERVALO_BATIDA = TRUE AND FTM1_CONTADOR_CICLO_BATIDA > 4 THEN
		FTM1_CONTADOR_CICLO_BATIDA := 1;
	END_IF
	
	
	//se o contador esta no ponto deste filtro e não esta no intervalo, liga saida
	IF FTM1_CONTADOR_CICLO_BATIDA = 1 AND NOT FTM1_LIBERA_INTERVALO_BATIDA  THEN
		SD_FLT11:=TRUE;
	ELSE
		SD_FLT11 := FALSE;
	END_IF

	//se o contador esta no ponto deste filtro e não esta no intervalo, liga saida
	IF FTM1_CONTADOR_CICLO_BATIDA = 2 AND NOT FTM1_LIBERA_INTERVALO_BATIDA  THEN
		SD_FLT12:=TRUE;
	ELSE
		SD_FLT12 := FALSE;
	END_IF

	//se o contador esta no ponto deste filtro e não esta no intervalo, liga saida
	IF FTM1_CONTADOR_CICLO_BATIDA = 3 AND NOT FTM1_LIBERA_INTERVALO_BATIDA  THEN
		SD_FLT13:=TRUE;
	ELSE
		SD_FLT13 := FALSE;
	END_IF

	//se o contador esta no ponto deste filtro e não esta no intervalo, liga saida
	IF FTM1_CONTADOR_CICLO_BATIDA = 4 AND NOT FTM1_LIBERA_INTERVALO_BATIDA  THEN
		SD_FLT14:=TRUE;
	ELSE
		SD_FLT14 := FALSE;
	END_IF
	
ELSE
	FTM1_CONTADOR_CICLO_BATIDA := 0;
	FTM1_LIBERA_BATIDA:=FALSE;
	FTM1_LIBERA_INTERVALO_BATIDA:= FALSE;
	SD_FLT11 := FALSE;
	SD_FLT12 := FALSE;
	SD_FLT13 := FALSE;
	SD_FLT14 := FALSE;
END_IF	


//Filtro de manga 2 ==================================================================
	IF BTS_FILTM2 = TRUE  AND AL_GERAL = FALSE   THEN
		IF LIGA_FTM2 = TRUE THEN
			LIGA_FTM2 := FALSE;
		ELSE
			LIGA_FTM2 := TRUE;
		END_IF
		BTS_FILTM2 := FALSE;
	ELSIF AL_GERAL = TRUE THEN  //delsiga em caso de alarme
		LIGA_FTM2 := FALSE;
		BTS_FILTM2 := FALSE;
	END_IF

//ciclo de batidas
IF LIGA_FTM2 THEN
		
	//condição para iniciar primeiro ciclo
	IF NOT FTM2_LIBERA_INTERVALO_BATIDA  AND NOT FTM2_LIBERA_BATIDA THEN	
		FTM2_LIBERA_BATIDA:=TRUE;
	END_IF
	
	//tempo de pulso da batida
	FTM2_TEMPO_BATIDA(IN:=FTM2_LIBERA_BATIDA, PT:= T#1S);
	
	//ao final do tempo vai para o intervalo e incrementa o contador de filtro
	IF FTM2_TEMPO_BATIDA.Q THEN
		FTM2_CONTADOR_CICLO_BATIDA := FTM2_CONTADOR_CICLO_BATIDA + 1;
		FTM2_LIBERA_INTERVALO_BATIDA := TRUE;
		FTM2_LIBERA_BATIDA:=FALSE;
	END_IF
	
	//tempo de intervalo para cada batida
	FTM2_TEMPO_INTERVALO_BATIDA(IN:=FTM2_LIBERA_INTERVALO_BATIDA, PT:= T#30S);
	
	//ao final tempo de intervalo, faz a batida
	IF FTM2_TEMPO_INTERVALO_BATIDA.Q  THEN
		FTM2_LIBERA_BATIDA:=TRUE;
		FTM2_LIBERA_INTERVALO_BATIDA:= FALSE;
	END_IF	
	
	//se chegou no filtro 4, reinicia o ciclo dos filtros 1 - 4
	IF FTM2_LIBERA_INTERVALO_BATIDA = TRUE AND FTM2_CONTADOR_CICLO_BATIDA > 4 THEN
		FTM2_CONTADOR_CICLO_BATIDA := 1;
	END_IF
	
	
	//se o contador esta no ponto deste filtro e não esta no intervalo, liga saida
	IF FTM2_CONTADOR_CICLO_BATIDA = 1 AND NOT FTM2_LIBERA_INTERVALO_BATIDA  THEN
		SD_FILT2123:=TRUE;
	ELSE
		SD_FILT2123 := FALSE;
	END_IF

	//se o contador esta no ponto deste filtro e não esta no intervalo, liga saida
	IF FTM2_CONTADOR_CICLO_BATIDA = 2 AND NOT FTM2_LIBERA_INTERVALO_BATIDA  THEN
		SD_FILT2224:=TRUE;
	ELSE
		SD_FILT2224 := FALSE;
	END_IF

	//se o contador esta no ponto deste filtro e não esta no intervalo, liga saida
	IF FTM2_CONTADOR_CICLO_BATIDA = 3 AND NOT FTM2_LIBERA_INTERVALO_BATIDA  THEN
		SD_FILT3133:=TRUE;
	ELSE
		SD_FILT3133 := FALSE;
	END_IF

	//se o contador esta no ponto deste filtro e não esta no intervalo, liga saida
	IF FTM2_CONTADOR_CICLO_BATIDA = 4 AND NOT FTM2_LIBERA_INTERVALO_BATIDA  THEN
		SD_FILT3234:=TRUE;
	ELSE
		SD_FILT3234 := FALSE;
	END_IF
	
ELSE
	FTM2_CONTADOR_CICLO_BATIDA := 0;
	FTM2_LIBERA_BATIDA:=FALSE;
	FTM2_LIBERA_INTERVALO_BATIDA:= FALSE;
	SD_FILT2123 := FALSE;
	SD_FILT2224 := FALSE;
	SD_FILT3133 := FALSE;
	SD_FILT3234 := FALSE;
END_IF

END_PROGRAM

// Device/Application/SA
PROGRAM SA
VAR

	//converte escala saida analogica 1 (bomba de baixa)
	converteSA1:LIN_TRAFO;
	//converte escala saida analogica 2 (bomba de alta 1)
	converteSA2:LIN_TRAFO;
	//converte escala saida analogica 3 (bomba de alta 2)
	converteSA3:LIN_TRAFO;
	//converte escala saida analogica 1 01 (bomba de perfume 1)	
	converteSA101:LIN_TRAFO;
	//converte escala saida analogica 2 01 (bomba de estrato)
	converteSA201:LIN_TRAFO;
	//converte escala saida analogica 3 01 (dosador 6)
	converteSA301:LIN_TRAFO;
	//converte escala saida analogica 4 01 (Exaustor 125 CV corrente)
	converteSA401:LIN_TRAFO;
	//converte escala saida analogica 1 02 (Exaustor 100 CV corrente)
	converteSA102:LIN_TRAFO;
	//converte escala saida analogica 2 02 (Bomba perfume 2)
	converteSA202:LIN_TRAFO;
	//converte escala saida analogica 3 02 (Ventilador Fluidizador)
	converteSA302:LIN_TRAFO;
	//converte escala saida analogica 4 02 (Queimador)
	converteSA402:LIN_TRAFO;
	
	
END_VAR

//NX6100

// Saida analógica 1 : NX6100 - Velocidade bomba de baixa  ( %) 
converteSA1(IN:=Vel_BB, IN_MIN:=0, IN_MAX:=100,OUT_MIN:=0, OUT_MAX:=4000);
SA1:= REAL_TO_INT(converteSA1.OUT);


// Saida analógica 2 : NX6100 - velocidade bomba de alta 1  (%) 
converteSA2(IN:=VEL_ALT1, IN_MIN:=0, IN_MAX:=100,OUT_MIN:=0, OUT_MAX:=4000);
SA2:= REAL_TO_INT(converteSA2.OUT);


// Saida analógica 3 : NX6100 - velocidade bomba de alta 2 ( %) 
converteSA3(IN:=VEL_ALT2, IN_MIN:=0, IN_MAX:=100,OUT_MIN:=0, OUT_MAX:=4000);
SA3:= REAL_TO_INT(converteSA3.OUT);


//NX6100_01
//=====================================================================================================================

// Saida analógica 1 : NX6100_01 - velocidade bomba de perfume 1 ( %) 
converteSA101(IN:=VEL_BP1, IN_MIN:=0, IN_MAX:=100,OUT_MIN:=0, OUT_MAX:=1000);
SA101:= REAL_TO_INT(converteSA101.OUT);

// Saida analógica 2 : NX6100_01 - velocidade Misturador Principal ( %) 
converteSA201(IN:=VEL_MPX, IN_MIN:=0, IN_MAX:=100,OUT_MIN:=0, OUT_MAX:=1000);
SA201:= REAL_TO_INT(converteSA201.OUT);

// Saida analógica 3 : NX6100_01 - Dosador 6 (0 - 100 hz) 
converteSA301(IN:=VEL_DSA6, IN_MIN:=0, IN_MAX:=100,OUT_MIN:=0, OUT_MAX:=4000);
SA301:= REAL_TO_INT(converteSA301.OUT);

// Saida analógica 4 : NX6100_01 - velocidade Exaustor 125 CV torre corrente ( %)  
converteSA401(IN:=Vel_EXTORRE, IN_MIN:=0, IN_MAX:=100,OUT_MIN:=0, OUT_MAX:=4000);
SA401:= REAL_TO_INT(converteSA401.OUT);

// NX6100_02
//======================================================================================================================

// Saida analógica 1 : NX6100_02 - velocidade ventilador queimador 100 CV corrente ( %) 
converteSA102(IN:=VEL_VENTQUEIMADOR, IN_MIN:=0, IN_MAX:=100,OUT_MIN:=0, OUT_MAX:=4000);
SA102:= REAL_TO_INT(converteSA102.OUT);

// Saida analógica 2 : NX6100_02 - velocidade bomba perfume 2 corrente ( %) 
converteSA202(IN:=VEL_BP2, IN_MIN:=0, IN_MAX:=100,OUT_MIN:=0, OUT_MAX:=1000);
SA202:= REAL_TO_INT(converteSA202.OUT);

// Saida analógica 3 : NX6100_02 - velocidade ventilador fluidizador corrente( %) 
converteSA302(IN:=PRST_VEL_VENTIFLUIDIZADOR, IN_MIN:=0, IN_MAX:=100,OUT_MIN:=0, OUT_MAX:=4000);
SA302:= REAL_TO_INT(converteSA302.OUT);

// Saida analógica 4 : NX6100_02 - queimador ( %) 
converteSA402(IN:=PRST_OLEO_QUEIMADOR, IN_MIN:=0, IN_MAX:=100,OUT_MIN:=0, OUT_MAX:=30000);
SA402:= REAL_TO_INT(converteSA402.OUT);

END_PROGRAM

// Device/Application/DSA1
PROGRAM DSA1
VAR
 	//Tempo de Homogenização em TIME
	TEMPO_DESLIGA_ZERAEVENTO:TON;
	//desliga botao limpa evento
	DESLIGA_BT_LIMPA_EVE:BOOL;
	//Liga Dosador manual
	LIGA_DS_MANUAL:BOOL;
	//Liga Dosador automatico
	LIGA_DS_AUTO:BOOL;
	//Espera o fluidizador baixar para o peso minino, pois atingiu o peso maximo
	ESPERA_FLUIDIZADOR_BAIXAR_PESO:BOOL;
	//Tempo desliga reset totalizador 1
	TMR_RESET_TOTAL1:TON;
	//Tempo desliga reset totalizador 2
	TMR_RESET_TOTAL2:TON;	
END_VAR

//POU relacionado aos comandos e alarmes do Dosador Gravimetrico 1 DEA-600 D-2B linha 1 (pó base 1)


//Controle manual PH 1

IF BTS_MAPH1 = FALSE THEN
//============================================================================
// comandos manuais 
//============================================================================	
	
	//Liga dosador 
	IF BTS_DS1 = TRUE AND AL_GERAL = FALSE THEN
		IF LIGA_DS_MANUAL = TRUE THEN
			LIGA_DS_MANUAL := FALSE;
		ELSE
			LIGA_DS_MANUAL :=TRUE;
		END_IF
		BTS_DS1 := FALSE;
	END_IF
	//desliga em caso de alarme
	IF AL_GERAL = TRUE THEN
		LIGA_DS_MANUAL := FALSE;
	END_IF
	
	//Calculo dosagem kg/h em manual
	PRST_VEL_DS1 := (PRST_VEL_PH1_MANUAL * 1000) * (PRST_PERC_DOSA_PB01 / 100);

	//em manual desliga comando do automatico
	LIGA_DS_AUTO := FALSE;
	
	
ELSE
//============================================================================
// comandos automatico
//============================================================================		
	
	//Liga dosador 
	IF  AL_GERAL = FALSE THEN
		LIGA_DS_AUTO :=TRUE;
	ELSE
		LIGA_DS_AUTO := FALSE;
	END_IF
	
	//zera velocidade do ph com peso maximo
	IF LEITURA_PESO_FLUI1 >= PRST_PESO_MAX_FLUID1 THEN
		ESPERA_FLUIDIZADOR_BAIXAR_PESO := TRUE;
	END_IF
	
	//ativa velocidade do ph com peso minimo
	IF LEITURA_PESO_FLUI1 <= PRST_PESO_MIN_FLUID1 THEN
		ESPERA_FLUIDIZADOR_BAIXAR_PESO := FALSE;
	END_IF
	
	
	IF ESPERA_FLUIDIZADOR_BAIXAR_PESO = FALSE THEN
		//Calculo dosagem kg/h em manual
		PRST_VEL_DS1 := (VELOCIDADE_PH1_AUTO) * (PRST_PERC_DOSA_PB01 / 100);
	ELSE
		PRST_VEL_DS1 := 0;
	END_IF
	
	
	//em auto desliga comando do manual
	LIGA_DS_MANUAL := FALSE;
END_IF

//Liga dosador
IF LIGA_DS_AUTO = TRUE OR LIGA_DS_MANUAL = TRUE THEN
	LIGA_DS1 := TRUE;
ELSE
	LIGA_DS1 := FALSE;
END_IF

//============================================================================
//  escrita da velocidade
//============================================================================

//Inversão da word da variavel da GVLPH: PRST_VEL_DS1, para variavel da GVLSCHENCK: PESO_DSA1
%QW15060 := %QW12772;
%QW15062 := %QW12770;


//============================================================================
// comandos 
//============================================================================

//conta tempo de homogenização
TEMPO_DESLIGA_ZERAEVENTO(IN:=BTS_LIMPEVE_DS1,PT:=T#10S);
DESLIGA_BT_LIMPA_EVE := TEMPO_DESLIGA_ZERAEVENTO.Q ;

IF DESLIGA_BT_LIMPA_EVE = TRUE THEN
	BTS_LIMPEVE_DS1 := FALSE;
END_IF


//bits de comando ============================================================
//Os bits de escrita inicio e parada da balança é invertido, por exemplo, para ligar o bit0 = false, e para parar o bit1=false
//Bit iniciar balança
IF LIGA_DS1 = FALSE THEN
	%QX15001.0 := FALSE;    //bit de ligar dosador, false para ativar		
ELSE
	%QX15001.0 := TRUE;		//bit de ligar dosador, true desativa	
END_IF

//bit parar balança
IF LIGA_DS1 = FALSE THEN
	%QX15001.1 := TRUE;		//bit de desligar dosador, true desativar
ELSE		
	%QX15001.1 := FALSE;	//bit de desligar dosador, false ativa	
END_IF

//bit limpar eventos
IF BTS_LIMPEVE_DS1 = TRUE THEN
	%QX15001.2 := TRUE;
ELSE
	%QX15001.2 := FALSE;
END_IF

//bit liberar
%QX15001.3 := TRUE;


//bit modo Volumetrico
IF BTS_MODVOL_DS1 = TRUE THEN
	%QX15001.4 := TRUE;	
ELSE
	%QX15001.4 := FALSE;
END_IF

//bit modo Gravimetrico
IF BTS_MODGRAV_DS1 = TRUE THEN
	%QX15001.5 := TRUE;	
ELSE
	%QX15001.5 := FALSE;
END_IF

//bit reinicializar Totalizador 1
IF BTS_ZERATOTAL1_DS1 = TRUE THEN
	%QX15001.6 := TRUE;
ELSE
	%QX15001.6 := FALSE;
END_IF

//Comando do Reset dos totalizadores geral, apontamento de producao
BTS_ZERATOTAL1_DS1 := BTS_RESET_TOTAL_SCHENCK;
//Tempo desliga reset totalizador 1
TMR_RESET_TOTAL1(IN:= BTS_ZERATOTAL1_DS1, PT:= T#15S);
//desliga o reset do totalizador ao zerar 
IF TMR_RESET_TOTAL1.Q = TRUE THEN
	BTS_ZERATOTAL1_DS1 := FALSE;
	BTS_RESET_TOTAL_SCHENCK := FALSE;
END_IF

//bit reinicializar Totalizador 2
IF BTS_ZERATOTAL2_DS1 = TRUE THEN
	%QX15001.7 := TRUE;
ELSE
	%QX15001.7 := FALSE;
END_IF
//Tempo desliga reset totalizador 2
TMR_RESET_TOTAL2(IN:= BTS_ZERATOTAL2_DS1, PT:= T#15S);
//desliga o reset do totalizador ao zerar 
IF TMR_RESET_TOTAL2.Q = TRUE THEN
	BTS_ZERATOTAL2_DS1 := FALSE;
END_IF

//bit Volume Sincrono
%QX15000.0 := TRUE;

//bit corre. umidade on
%QX15000.1 := TRUE;

//bit corre. umidade off
%QX15000.2 := TRUE;

//bit acionamento med. off
%QX15000.3 := TRUE;

//bit retorno da comporta PMS
%QX15000.4 := TRUE;

//bit reservado
%QX15000.5 := TRUE;

//bit reservado
%QX15000.6 := TRUE;

//bit reservado
%QX15000.7 := TRUE;


//====================================================================================
// Leitura Valores REAL 
//====================================================================================

//Totalizador1, leitura em Kg, 
//Inversão da word da variavel da GVLSCHENCK: LEITURA_TOTALIZADOR1_DSA1, para variavel da GVLPH: TOTALIZADOR1_KG 
%QW10000 := %IW15132;
%QW10002 := %IW15130;

//Totalizador2, leitura em Kg, apenas invertidos as words
//Inversão da word da variavel da GVLSCHENCK: LEITURA_TOTALIZADOR2_DSA1, para variavel da GVLPH: TOTALIZADOR2_KG 
%QW10004 := %IW15192;
%QW10006 := %IW15190;

//Totalizador3, leitura em Tonelada, invertidos as words e dividido por 1000 
//Inversão da word da variavel da GVLSCHENCK: LEITURA_TOTALIZADOR3_DSA1, para variavel da GVLPH: TOTALIZADOR3_KG 
%QW10008 := %IW15302;
%QW10010 := %IW15300;
TOTALIZADOR3_TON_DS1 := TOTALIZADOR3_KG_DS1 / 1000;

//Velocidade atual do dosador
%QW10300 := %IW15252;
%QW10302 := %IW15250;

VELOCIDADE_REAL_DS1 := VELOCIDADE_REAL2_DS1 ;

END_PROGRAM

// Device/Application/DSA2
PROGRAM DSA2
VAR
	//Tempo de Homogenização em TIME
	TEMPO_DESLIGA_ZERAEVENTO:TON;
	//desliga botao limpa evento
	DESLIGA_BT_LIMPA_EVE:BOOL;
	//Liga Dosador manual
	LIGA_DS_MANUAL:BOOL;
	//Liga Dosador automatico
	LIGA_DS_AUTO:BOOL;
	//Espera o fluidizador baixar para o peso minino, pois atingiu o peso maximo
	ESPERA_FLUIDIZADOR_BAIXAR_PESO:BOOL;
	//Tempo desliga reset totalizador 1
	TMR_RESET_TOTAL1:TON;
	//Tempo desliga reset totalizador 2
	TMR_RESET_TOTAL2:TON;
END_VAR

//POU relacionado aos comandos e alarmes do Dosador Gravimetrico 2 DEA-300 D-4B linha 1

// Controle manual dos equipamentos 
//=================================================================================================

//Controle manual PH 1

IF BTS_MAPH1 = FALSE THEN
//============================================================================
// comandos manuais 
//============================================================================	
	
	//Liga dosador 
	IF BTS_DS2 = TRUE AND AL_GERAL = FALSE THEN
		IF LIGA_DS_MANUAL = TRUE THEN
			LIGA_DS_MANUAL := FALSE;
		ELSE
			LIGA_DS_MANUAL :=TRUE;
		END_IF
		BTS_DS2 := FALSE;
	END_IF
	//desliga em caso de alarme
	IF AL_GERAL = TRUE THEN
		LIGA_DS_MANUAL := FALSE;
	END_IF

	//Calculo dosagem kg/h em manual
	PRST_VEL_DS2 := (PRST_VEL_PH1_MANUAL * 1000) * (PRST_PERC_DOSA_DS02 / 100);
	
	//em manual desliga comando do automatico
	LIGA_DS_AUTO := FALSE;
	
ELSE
//============================================================================
// comandos automatico
//============================================================================		
	
	//Liga dosador 
	IF  AL_GERAL = FALSE THEN
		LIGA_DS_AUTO :=TRUE;
	ELSE
		LIGA_DS_AUTO := FALSE;
	END_IF
	
		//zera velocidade do ph com peso maximo
	IF LEITURA_PESO_FLUI1 >= PRST_PESO_MAX_FLUID1 THEN
		ESPERA_FLUIDIZADOR_BAIXAR_PESO := TRUE;
	END_IF
	
	//ativa velocidade do ph com peso minimo
	IF LEITURA_PESO_FLUI1 <= PRST_PESO_MIN_FLUID1 THEN
		ESPERA_FLUIDIZADOR_BAIXAR_PESO := FALSE;
	END_IF
	
	IF ESPERA_FLUIDIZADOR_BAIXAR_PESO = FALSE THEN
		//Calculo dosagem kg/h em manual
		PRST_VEL_DS2 := (VELOCIDADE_PH1_AUTO) * (PRST_PERC_DOSA_DS02 / 100);
	ELSE
		PRST_VEL_DS2 := 0;
	END_IF
	
	//em auto desliga comando do manual
	LIGA_DS_MANUAL := FALSE;
	
END_IF

//Liga dosador
IF LIGA_DS_AUTO = TRUE OR LIGA_DS_MANUAL = TRUE THEN
	LIGA_DS2 := TRUE;
ELSE
	LIGA_DS2 := FALSE;
END_IF

//============================================================================
//  escrita da velocidade
//============================================================================

//Inversão da word da variavel da GVLPH: PRST_VEL_DS2, para variavel da GVLSCHENCK: PESO_DSA2
%QW15064 := %QW12728;
%QW15066 := %QW12726;

//============================================================================
// comandos que independem do comando manual/auto
//============================================================================

//conta tempo de homogenização
TEMPO_DESLIGA_ZERAEVENTO(IN:=BTS_LIMPEVE_DS2,PT:=T#10S);
DESLIGA_BT_LIMPA_EVE := TEMPO_DESLIGA_ZERAEVENTO.Q ;

IF DESLIGA_BT_LIMPA_EVE = TRUE THEN
	BTS_LIMPEVE_DS2 := FALSE;
END_IF

//bits de comando ============================================================
//Os bits de escrita inicio e parada da balança é invertido, por exemplo, para ligar o bit0 = false, e para parar o bit1=false

//Bit iniciar balança
IF LIGA_DS2 = FALSE THEN
	%QX15003.0 := FALSE;    //bit de ligar dosador, false para ativar	
ELSE
	%QX15003.0 := TRUE;		//bit de ligar dosador, true desativa	
END_IF

//bit parar balança
IF LIGA_DS2 = FALSE THEN
	%QX15003.1 := TRUE;		//bit de desligar dosador, true desativar
ELSE		
	%QX15003.1 := FALSE;	//bit de desligar dosador, false ativa	
END_IF

//bit limpar eventos
IF BTS_LIMPEVE_DS2 = TRUE THEN
	%QX15003.2 := TRUE;
ELSE
	%QX15003.2 := FALSE;
END_IF

//bit liberar
%QX15003.3 := TRUE;

//bit modo Volumetrico
IF BTS_MODVOL_DS2 = TRUE THEN
	%QX15003.4 := TRUE;
ELSE
	%QX15003.4 := FALSE;
END_IF
	
//bit modo Gravimetrico
IF BTS_MODGRAV_DS2 = TRUE THEN
	%QX15003.5 := TRUE;
ELSE
	%QX15003.5 := FALSE;
END_IF

//bit reinicializar Totalizador 1
IF BTS_ZERATOTAL1_DS2 = TRUE THEN
	%QX15003.6 := TRUE;
ELSE
	%QX15003.6 := FALSE;
END_IF

//Comando do Reset dos totalizadores geral, apontamento de producao
BTS_ZERATOTAL1_DS2 := BTS_RESET_TOTAL_SCHENCK;
//Tempo desliga reset totalizador 1
TMR_RESET_TOTAL1(IN:= BTS_ZERATOTAL1_DS2, PT:= T#15S);
//desliga o reset do totalizador ao zerar 
IF TMR_RESET_TOTAL1.Q = TRUE THEN
	BTS_ZERATOTAL1_DS2 := FALSE;
	BTS_RESET_TOTAL_SCHENCK := FALSE;
END_IF

//bit reinicializar Totalizador 2
IF BTS_ZERATOTAL2_DS2 = TRUE THEN
	%QX15003.7 := TRUE;
ELSE
	%QX15003.7 := FALSE;
END_IF
//Tempo desliga reset totalizador 2
TMR_RESET_TOTAL2(IN:= BTS_ZERATOTAL2_DS2, PT:= T#15S);
//desliga o reset do totalizador ao zerar 
IF TMR_RESET_TOTAL2.Q = TRUE THEN
	BTS_ZERATOTAL2_DS2 := FALSE;
END_IF

//bit Volume Sincrono
%QX15002.0 := TRUE;

//bit corre. umidade on
%QX15002.1 := TRUE;

//bit corre. umidade off
%QX15002.2 := TRUE;

//bit acionamento med. off
%QX15002.3 := TRUE;

//bit retorno da comporta PMS
%QX15002.4 := TRUE;

//bit reservado
%QX15002.5 := TRUE;

//bit reservado
%QX15002.6 := TRUE;

//bit reservado
%QX15002.7 := TRUE;


//====================================================================================
// Leitura Valores REAL 
//====================================================================================

//Totalizador1, leitura em Kg, 
//Inversão da word da variavel da GVLSCHENCK: LEITURA_TOTALIZADOR1_DSA2, para variavel da GVLPH: TOTALIZADOR1_KG 
%QW10016 := %IW15136;
%QW10018 := %IW15134;

//Totalizador2, leitura em Kg, apenas invertidos as words
//Inversão da word da variavel da GVLSCHENCK: LEITURA_TOTALIZADOR2_DSA2, para variavel da GVLPH: TOTALIZADOR2_KG 
%QW10020 := %IW15196;
%QW10022 := %IW15194;

//Totalizador3, leitura em Tonelada, invertidos as words e dividido por 1000 
//Inversão da word da variavel da GVLSCHENCK: LEITURA_TOTALIZADOR3_DSA2, para variavel da GVLPH: TOTALIZADOR3_KG 
%QW10024 := %IW15306;
%QW10026 := %IW15304;
TOTALIZADOR3_TON_DS2 := TOTALIZADOR3_KG_DS2 / 1000;

//Velocidade atual do dosador
%QW10304 := %IW15256;
%QW10306 := %IW15254;

VELOCIDADE_REAL_DS2 := VELOCIDADE_REAL2_DS2;

END_PROGRAM

// Device/Application/DSA3
PROGRAM DSA3
VAR
	//Tempo de Homogenização em TIME
	TEMPO_DESLIGA_ZERAEVENTO:TON;
	//desliga botao limpa evento
	DESLIGA_BT_LIMPA_EVE:BOOL;
	//Liga Dosador manual
	LIGA_DS_MANUAL:BOOL;
	//Liga Dosador automatico
	LIGA_DS_AUTO:BOOL;
	//Espera o fluidizador baixar para o peso minino, pois atingiu o peso maximo
	ESPERA_FLUIDIZADOR_BAIXAR_PESO:BOOL;
	//Tempo desliga reset totalizador 1
	TMR_RESET_TOTAL1:TON;
	//Tempo desliga reset totalizador 2
	TMR_RESET_TOTAL2:TON;
END_VAR

//POU relacionado aos comandos e alarmes do Dosador Gravimetrico 3 DEA-300 D-3B linha 1


//Controle manual PH 1

IF BTS_MAPH1 = FALSE THEN
//============================================================================
// comandos manuais 
//============================================================================	
	
	//Liga dosador 
	IF BTS_DS3 = TRUE AND AL_GERAL = FALSE THEN
		IF LIGA_DS_MANUAL = TRUE THEN
			LIGA_DS_MANUAL := FALSE;
		ELSE
			LIGA_DS_MANUAL :=TRUE;
		END_IF
		BTS_DS3 := FALSE;
	END_IF
	//desliga em caso de alarme
	IF AL_GERAL = TRUE THEN
		LIGA_DS_MANUAL := FALSE;
	END_IF
	
	//Calculo dosagem kg/h em manual
	PRST_VEL_DS3 := (PRST_VEL_PH1_MANUAL * 1000) * (PRST_PERC_DOSA_DS03 / 100);

	//em manual desliga comando do automatico
	LIGA_DS_AUTO := FALSE;
	
ELSE
//============================================================================
// comandos automatico
//============================================================================		
	
	//Liga dosador 
	IF  AL_GERAL = FALSE THEN
		LIGA_DS_AUTO :=TRUE;
	ELSE
		LIGA_DS_AUTO := FALSE;
	END_IF
	
	//zera velocidade do ph com peso maximo
	IF LEITURA_PESO_FLUI1 >= PRST_PESO_MAX_FLUID1 THEN
		ESPERA_FLUIDIZADOR_BAIXAR_PESO := TRUE;
	END_IF
	
	//ativa velocidade do ph com peso minimo
	IF LEITURA_PESO_FLUI1 <= PRST_PESO_MIN_FLUID1 THEN
		ESPERA_FLUIDIZADOR_BAIXAR_PESO := FALSE;
	END_IF
	
	IF ESPERA_FLUIDIZADOR_BAIXAR_PESO = FALSE THEN
		//Calculo dosagem kg/h em manual
		PRST_VEL_DS3 := (VELOCIDADE_PH1_AUTO) * (PRST_PERC_DOSA_DS03 / 100);
	ELSE
		PRST_VEL_DS3 := 0;
	END_IF
	
	//em auto desliga comando do manual
	LIGA_DS_MANUAL := FALSE;
	
END_IF

//Liga dosador
IF LIGA_DS_AUTO = TRUE OR LIGA_DS_MANUAL = TRUE THEN
	LIGA_DS3 := TRUE;
ELSE
	LIGA_DS3 := FALSE;
END_IF


//============================================================================
//  escrita da velocidade
//============================================================================

//Inversão da word da variavel da GVLPH: PRST_VEL_DS3, para variavel da GVLSCHENCK: PESO_DSA3
%QW15068 := %QW12732;
%QW15070 := %QW12730;


//============================================================================
// comandos que independem do comando manual/auto
//============================================================================
//conta tempo de homogenização
TEMPO_DESLIGA_ZERAEVENTO(IN:=BTS_LIMPEVE_DS3,PT:=T#10S);
DESLIGA_BT_LIMPA_EVE := TEMPO_DESLIGA_ZERAEVENTO.Q ;

IF DESLIGA_BT_LIMPA_EVE = TRUE THEN
	BTS_LIMPEVE_DS3 := FALSE;
END_IF

//bits de comando ============================================================
//Os bits de escrita inicio e parada da balança é invertido, por exemplo, para ligar o bit0 = false, e para parar o bit1=false

//Bit iniciar balança
IF LIGA_DS3 = FALSE THEN
	%QX15005.0 := FALSE;    //bit de ligar dosador, false para ativar	
ELSE
	%QX15005.0 := TRUE;		//bit de ligar dosador, true desativa	
END_IF

//bit parar balança
IF LIGA_DS3 = FALSE THEN
	%QX15005.1 := TRUE;		//bit de desligar dosador, true desativar
ELSE		
	%QX15005.1 := FALSE;	//bit de desligar dosador, false ativa	
END_IF

//bit limpar eventos
IF BTS_LIMPEVE_DS3 = TRUE THEN
	%QX15005.2 := TRUE;
ELSE
	%QX15005.2 := FALSE;
END_IF

//bit liberar
%QX15005.3 := TRUE;

//bit modo Volumetrico
IF BTS_MODVOL_DS3 = TRUE THEN
	%QX15005.4 := TRUE;
ELSE
	%QX15005.4 := FALSE;
END_IF
	
//bit modo Gravimetrico
IF BTS_MODGRAV_DS3 = TRUE THEN
	%QX15005.5 := TRUE;
ELSE
	%QX15005.5 := FALSE;
END_IF

//bit reinicializar Totalizador 1
IF BTS_ZERATOTAL1_DS3 = TRUE THEN
	%QX15005.6 := TRUE;
ELSE
	%QX15005.6 := FALSE;
END_IF

//Comando do Reset dos totalizadores geral, apontamento de producao
BTS_ZERATOTAL1_DS3 := BTS_RESET_TOTAL_SCHENCK;
//Tempo desliga reset totalizador 1
TMR_RESET_TOTAL1(IN:= BTS_ZERATOTAL1_DS3, PT:= T#15S);
//desliga o reset do totalizador ao zerar 
IF TMR_RESET_TOTAL1.Q = TRUE THEN
	BTS_ZERATOTAL1_DS3 := FALSE;
	BTS_RESET_TOTAL_SCHENCK := FALSE;
END_IF

//bit reinicializar Totalizador 2
IF BTS_ZERATOTAL2_DS3 = TRUE THEN
	%QX15005.7 := TRUE;
ELSE
	%QX15005.7 := FALSE;
END_IF
//Tempo desliga reset totalizador 2
TMR_RESET_TOTAL2(IN:= BTS_ZERATOTAL2_DS3, PT:= T#15S);
//desliga o reset do totalizador ao zerar 
IF TMR_RESET_TOTAL2.Q = TRUE THEN
	BTS_ZERATOTAL2_DS3 := FALSE;
END_IF


//bit Volume Sincrono
%QX15004.0 := TRUE;

//bit corre. umidade on
%QX15004.1 := TRUE;

//bit corre. umidade off
%QX15004.2 := TRUE;

//bit acionamento med. off
%QX15004.3 := TRUE;

//bit retorno da comporta PMS
%QX15004.4 := TRUE;

//bit reservado
%QX15004.5 := TRUE;

//bit reservado
%QX15004.6 := TRUE;

//bit reservado
%QX15004.7 := TRUE;


//====================================================================================
// Leitura Valores REAL 
//====================================================================================

//Totalizador1, leitura em Kg, 
//Inversão da word da variavel da GVLSCHENCK: LEITURA_TOTALIZADOR1_DSA3, para variavel da GVLPH: TOTALIZADOR1_KG 
%QW10032 := %IW15140;
%QW10034 := %IW15138;

//Totalizador2, leitura em Kg, apenas invertidos as words
//Inversão da word da variavel da GVLSCHENCK: LEITURA_TOTALIZADOR2_DSA3, para variavel da GVLPH: TOTALIZADOR2_KG 
%QW10036 := %IW15200;
%QW10038 := %IW15198;

//Totalizador3, leitura em Tonelada, invertidos as words e dividido por 1000 
//Inversão da word da variavel da GVLSCHENCK: LEITURA_TOTALIZADOR3_DSA3, para variavel da GVLPH: TOTALIZADOR3_KG 
%QW10040 := %IW15310;
%QW10042 := %IW15308;
TOTALIZADOR3_TON_DS3 := TOTALIZADOR3_KG_DS3 / 1000;

//Velocidade atual do dosador
%QW10308 := %IW15260;
%QW10310 := %IW15258;

VELOCIDADE_REAL_DS3 := VELOCIDADE_REAL2_DS3 ;

END_PROGRAM

// Device/Application/DSA4
PROGRAM DSA4
VAR
	//Tempo de Homogenização em TIME
	TEMPO_DESLIGA_ZERAEVENTO:TON;
	//desliga botao limpa evento
	DESLIGA_BT_LIMPA_EVE:BOOL;
	//Liga Dosador manual
	LIGA_DS_MANUAL:BOOL;
	//Liga Dosador automatico
	LIGA_DS_AUTO:BOOL;
	//Espera o fluidizador baixar para o peso minino, pois atingiu o peso maximo
	ESPERA_FLUIDIZADOR_BAIXAR_PESO:BOOL;
		//Tempo desliga reset totalizador 1
	TMR_RESET_TOTAL1:TON;
	//Tempo desliga reset totalizador 2
	TMR_RESET_TOTAL2:TON;
END_VAR

//POU relacionado aos comandos e alarmes do Dosador Gravimetrico 4 MECHATRON D-6B linha 1


//Controle manual PH 1

IF BTS_MAPH1 = FALSE THEN
//============================================================================
// comandos manuais 
//============================================================================	
	
	//Liga dosador 
	IF BTS_DS4 = TRUE AND AL_GERAL = FALSE THEN
		IF LIGA_DS_MANUAL = TRUE THEN
			LIGA_DS_MANUAL := FALSE;
		ELSE
			LIGA_DS_MANUAL :=TRUE;
		END_IF
		BTS_DS4 := FALSE;
	END_IF
	//desliga em caso de alarme
	IF AL_GERAL = TRUE THEN
		LIGA_DS_MANUAL := FALSE;
	END_IF

	//Calculo dosagem kg/h em manual
	PRST_VEL_DS4 := (PRST_VEL_PH1_MANUAL * 1000) * (PRST_PERC_DOSA_DS04 / 100);
	
	//em manual desliga comando do automatico
	LIGA_DS_AUTO := FALSE;
ELSE
//============================================================================
// comandos automatico
//============================================================================		
	
	//Liga dosador 
	IF  AL_GERAL = FALSE THEN
		LIGA_DS_AUTO :=TRUE;
	ELSE
		LIGA_DS_AUTO := FALSE;
	END_IF
	
	//zera velocidade do ph com peso maximo
	IF LEITURA_PESO_FLUI1 >= PRST_PESO_MAX_FLUID1 THEN
		ESPERA_FLUIDIZADOR_BAIXAR_PESO := TRUE;
	END_IF
	
	//ativa velocidade do ph com peso minimo
	IF LEITURA_PESO_FLUI1 <= PRST_PESO_MIN_FLUID1 THEN
		ESPERA_FLUIDIZADOR_BAIXAR_PESO := FALSE;
	END_IF
	
	IF ESPERA_FLUIDIZADOR_BAIXAR_PESO = FALSE THEN
		//Calculo dosagem kg/h em manual
		PRST_VEL_DS4 := (VELOCIDADE_PH1_AUTO) * (PRST_PERC_DOSA_DS04 / 100);
	ELSE
		PRST_VEL_DS4 := 0;
	END_IF
	
	//em auto desliga comando do manual
	LIGA_DS_MANUAL := FALSE;
END_IF

//Liga dosador
IF LIGA_DS_AUTO = TRUE OR LIGA_DS_MANUAL = TRUE THEN
	LIGA_DS4 := TRUE;
ELSE
	LIGA_DS4 := FALSE;
END_IF



//============================================================================
//  escrita da velocidade
//============================================================================

//Inversão da word da variavel da GVLPH: PRST_VEL_DS4, para variavel da GVLSCHENCK: PESO_DSA4
%QW15072 := %QW12736;
%QW15074 := %QW12734;

//============================================================================
// comandos que independem do comando manual/auto
//============================================================================

//conta tempo de homogenização
TEMPO_DESLIGA_ZERAEVENTO(IN:=BTS_LIMPEVE_DS4,PT:=T#10S);
DESLIGA_BT_LIMPA_EVE := TEMPO_DESLIGA_ZERAEVENTO.Q ;

IF DESLIGA_BT_LIMPA_EVE = TRUE THEN
	BTS_LIMPEVE_DS4 := FALSE;
END_IF

//bits de comando ============================================================
//Os bits de escrita inicio e parada da balança é invertido, por exemplo, para ligar o bit0 = false, e para parar o bit1=false

//Bit iniciar balança
IF LIGA_DS4 = FALSE THEN
	%QX15007.0 := FALSE;    //bit de ligar dosador, false para ativar	
ELSE
	%QX15007.0 := TRUE;		//bit de ligar dosador, true desativa	
END_IF

//bit parar balança
IF LIGA_DS4 = FALSE THEN
	%QX15007.1 := TRUE;		//bit de desligar dosador, true desativar
ELSE		
	%QX15007.1 := FALSE;	//bit de desligar dosador, false ativa	
END_IF

//bit limpar eventos
IF BTS_LIMPEVE_DS4 = TRUE THEN
	%QX15007.2 := TRUE;
ELSE
	%QX15007.2 := FALSE;
END_IF

//bit liberar
%QX15007.3 := TRUE;

//bit modo Volumetrico
IF BTS_MODVOL_DS4 = TRUE THEN
	%QX15007.4 := TRUE;
ELSE
	%QX15007.4 := FALSE;
END_IF
	
//bit modo Gravimetrico
IF BTS_MODGRAV_DS4 = TRUE THEN
	%QX15007.5 := TRUE;
ELSE
	%QX15007.5 := FALSE;
END_IF

//bit reinicializar Totalizador 1
IF BTS_ZERATOTAL1_DS4 = TRUE THEN
	%QX15007.6 := TRUE;
ELSE
	%QX15007.6 := FALSE;
END_IF

//Comando do Reset dos totalizadores geral, apontamento de producao
BTS_ZERATOTAL1_DS4 := BTS_RESET_TOTAL_SCHENCK;
//Tempo desliga reset totalizador 1
TMR_RESET_TOTAL1(IN:= BTS_ZERATOTAL1_DS4, PT:= T#15S);
//desliga o reset do totalizador ao zerar 
IF TMR_RESET_TOTAL1.Q = TRUE THEN
	BTS_ZERATOTAL1_DS4 := FALSE;
	BTS_RESET_TOTAL_SCHENCK := FALSE;
END_IF

//bit reinicializar Totalizador 2
IF BTS_ZERATOTAL2_DS4 = TRUE THEN
	%QX15007.7 := TRUE;
ELSE
	%QX15007.7 := FALSE;
END_IF
//Tempo desliga reset totalizador 2
TMR_RESET_TOTAL2(IN:= BTS_ZERATOTAL2_DS4, PT:= T#15S);
//desliga o reset do totalizador ao zerar 
IF TMR_RESET_TOTAL2.Q = TRUE THEN
	BTS_ZERATOTAL2_DS4 := FALSE;
END_IF

//bit Volume Sincrono
%QX15006.0 := TRUE;

//bit corre. umidade on
%QX15006.1 := TRUE;

//bit corre. umidade off
%QX15006.2 := TRUE;

//bit acionamento med. off
%QX15006.3 := TRUE;

//bit retorno da comporta PMS
%QX15006.4 := TRUE;

//bit reservado
%QX15006.5 := TRUE;

//bit reservado
%QX15006.6 := TRUE;

//bit reservado
%QX15006.7 := TRUE;


//====================================================================================
// Leitura Valores REAL 
//====================================================================================

//Totalizador1, leitura em Kg, 
//Inversão da word da variavel da GVLSCHENCK: LEITURA_TOTALIZADOR1_DSA4, para variavel da GVLPH: TOTALIZADOR1_KG 
%QW10048 := %IW15144;
%QW10050 := %IW15142;

//Totalizador2, leitura em Kg, apenas invertidos as words
//Inversão da word da variavel da GVLSCHENCK: LEITURA_TOTALIZADOR2_DSA4, para variavel da GVLPH: TOTALIZADOR2_KG 
%QW10052 := %IW15204;
%QW10054 := %IW15202;

//Totalizador3, leitura em Tonelada, invertidos as words e dividido por 1000 
//Inversão da word da variavel da GVLSCHENCK: LEITURA_TOTALIZADOR3_DSA4, para variavel da GVLPH: TOTALIZADOR3_KG 
%QW10056 := %IW15314;
%QW10058 := %IW15312;
TOTALIZADOR3_TON_DS4 := TOTALIZADOR3_KG_DS4 / 1000;

//Velocidade atual do dosador
%QW10312 := %IW15264;
%QW10314 := %IW15262;

VELOCIDADE_REAL_DS4 := VELOCIDADE_REAL2_DS4 ;

END_PROGRAM

// Device/Application/DSA5
PROGRAM DSA5
VAR
	//Tempo de Homogenização em TIME
	TEMPO_DESLIGA_ZERAEVENTO:TON;
	//desliga botao limpa evento
	DESLIGA_BT_LIMPA_EVE:BOOL;
	//Liga Dosador manual
	LIGA_DS_MANUAL:BOOL;
	//Liga Dosador automatico
	LIGA_DS_AUTO:BOOL;
	//Espera o fluidizador baixar para o peso minino, pois atingiu o peso maximo
	ESPERA_FLUIDIZADOR_BAIXAR_PESO:BOOL;
	//Tempo desliga reset totalizador 1
	TMR_RESET_TOTAL1:TON;
	//Tempo desliga reset totalizador 2
	TMR_RESET_TOTAL2:TON;
END_VAR

//POU relacionado aos comandos e alarmes do Dosador Gravimetrico 5 MECHATRON D-7B linha 1


//Controle manual PH 1

IF BTS_MAPH1 = FALSE THEN
//============================================================================
// comandos manuais 
//============================================================================	
	
	//Liga dosador 
	IF BTS_DS5 = TRUE AND AL_GERAL = FALSE THEN
		IF LIGA_DS_MANUAL = TRUE THEN
			LIGA_DS_MANUAL := FALSE;
		ELSE
			LIGA_DS_MANUAL :=TRUE;
		END_IF
		BTS_DS5 := FALSE;
	END_IF
	//desliga em caso de alarme
	IF AL_GERAL = TRUE THEN
		LIGA_DS_MANUAL := FALSE;
	END_IF
	
	//Calculo dosagem kg/h em manual
	PRST_VEL_DS5 := (PRST_VEL_PH1_MANUAL * 1000) * (PRST_PERC_DOSA_DS05 / 100);

	//em manual desliga comando do automatico
	LIGA_DS_AUTO := FALSE;
ELSE
//============================================================================
// comandos automatico
//============================================================================		
	
	//Liga dosador 
	IF  AL_GERAL = FALSE THEN
		LIGA_DS_AUTO :=TRUE;
	ELSE
		LIGA_DS_AUTO := FALSE;
	END_IF
	
	//zera velocidade do ph com peso maximo
	IF LEITURA_PESO_FLUI1 >= PRST_PESO_MAX_FLUID1 THEN
		ESPERA_FLUIDIZADOR_BAIXAR_PESO := TRUE;
	END_IF
	
	//ativa velocidade do ph com peso minimo
	IF LEITURA_PESO_FLUI1 <= PRST_PESO_MIN_FLUID1 THEN
		ESPERA_FLUIDIZADOR_BAIXAR_PESO := FALSE;
	END_IF
	
	IF ESPERA_FLUIDIZADOR_BAIXAR_PESO = FALSE THEN
		//Calculo dosagem kg/h em manual
		PRST_VEL_DS5 := (VELOCIDADE_PH1_AUTO) * (PRST_PERC_DOSA_DS05 / 100);
	ELSE
		PRST_VEL_DS5 := 0;
	END_IF
	
	
	//em auto desliga comando do manual
	LIGA_DS_MANUAL := FALSE;
END_IF

//Liga dosador
IF LIGA_DS_AUTO = TRUE OR LIGA_DS_MANUAL = TRUE THEN
	LIGA_DS5 := TRUE;
ELSE
	LIGA_DS5 := FALSE;
END_IF

//============================================================================
//  escrita da velocidade
//============================================================================

//Inversão da word da variavel da GVLPH: PRST_VEL_DS5, para variavel da GVLSCHENCK: PESO_DSA5
%QW15076 := %QW12740;
%QW15078 := %QW12738;

//============================================================================
// comandos que independem do comando manual/auto
//============================================================================

//conta tempo de homogenização
TEMPO_DESLIGA_ZERAEVENTO(IN:=BTS_LIMPEVE_DS5,PT:=T#10S);
DESLIGA_BT_LIMPA_EVE := TEMPO_DESLIGA_ZERAEVENTO.Q ;

IF DESLIGA_BT_LIMPA_EVE = TRUE THEN
	BTS_LIMPEVE_DS5 := FALSE;
END_IF

//bits de comando ============================================================
//Os bits de escrita inicio e parada da balança é invertido, por exemplo, para ligar o bit0 = false, e para parar o bit1=false

//Bit iniciar balança
IF LIGA_DS5 = FALSE THEN
	%QX15009.0 := FALSE;    //bit de ligar dosador, false para ativar	
ELSE
	%QX15009.0 := TRUE;		//bit de ligar dosador, true desativa	
END_IF

//bit parar balança
IF LIGA_DS5 = FALSE THEN
	%QX15009.1 := TRUE;		//bit de desligar dosador, true desativar
ELSE		
	%QX15009.1 := FALSE;	//bit de desligar dosador, false ativa	
END_IF

//bit limpar eventos
IF BTS_LIMPEVE_DS5 = TRUE THEN
	%QX15009.2 := TRUE;
ELSE
	%QX15009.2 := FALSE;
END_IF

//bit liberar
%QX15009.3 := TRUE;

//bit modo Volumetrico
IF BTS_MODVOL_DS5 = TRUE THEN
	%QX15009.4 := TRUE;
ELSE
	%QX15009.4 := FALSE;
END_IF
	
//bit modo Gravimetrico
IF BTS_MODGRAV_DS5 = TRUE THEN
	%QX15009.5 := TRUE;
ELSE
	%QX15009.5 := FALSE;
END_IF

//bit reinicializar Totalizador 1
IF BTS_ZERATOTAL1_DS5 = TRUE THEN
	%QX15009.6 := TRUE;
ELSE
	%QX15009.6 := FALSE;
END_IF

//Comando do Reset dos totalizadores geral, apontamento de producao
BTS_ZERATOTAL1_DS5 := BTS_RESET_TOTAL_SCHENCK;
//Tempo desliga reset totalizador 1
TMR_RESET_TOTAL1(IN:= BTS_ZERATOTAL1_DS5, PT:= T#15S);
//desliga o reset do totalizador ao zerar 
IF TMR_RESET_TOTAL1.Q = TRUE THEN
	BTS_ZERATOTAL1_DS5 := FALSE;
	BTS_RESET_TOTAL_SCHENCK := FALSE;
END_IF

//bit reinicializar Totalizador 2
IF BTS_ZERATOTAL2_DS5 = TRUE THEN
	%QX15009.7 := TRUE;
ELSE
	%QX15009.7 := FALSE;
END_IF
//Tempo desliga reset totalizador 2
TMR_RESET_TOTAL2(IN:= BTS_ZERATOTAL2_DS5, PT:= T#15S);
//desliga o reset do totalizador ao zerar 
IF TMR_RESET_TOTAL2.Q = TRUE THEN
	BTS_ZERATOTAL2_DS5 := FALSE;
END_IF

//bit Volume Sincrono
%QX15008.0 := TRUE;

//bit corre. umidade on
%QX15008.1 := TRUE;

//bit corre. umidade off
%QX15008.2 := TRUE;

//bit acionamento med. off
%QX15008.3 := TRUE;

//bit retorno da comporta PMS
%QX15008.4 := TRUE;

//bit reservado
%QX15008.5 := TRUE;

//bit reservado
%QX15008.6 := TRUE;

//bit reservado
%QX15008.7 := TRUE;


//====================================================================================
// Leitura Valores REAL 
//====================================================================================

//Totalizador1, leitura em Kg, 
//Inversão da word da variavel da GVLSCHENCK: LEITURA_TOTALIZADOR1_DSA5, para variavel da GVLPH: TOTALIZADOR1_KG 
%QW10064 := %IW15148;
%QW10066 := %IW15146;

//Totalizador2, leitura em Kg, apenas invertidos as words
//Inversão da word da variavel da GVLSCHENCK: LEITURA_TOTALIZADOR2_DSA5, para variavel da GVLPH: TOTALIZADOR2_KG 
%QW10068 := %IW15208;
%QW10070 := %IW15206;

//Totalizador3, leitura em Tonelada, invertidos as words e dividido por 1000 
//Inversão da word da variavel da GVLSCHENCK: LEITURA_TOTALIZADOR3_DSA5, para variavel da GVLPH: TOTALIZADOR3_KG 
%QW10072 := %IW15318;
%QW10074 := %IW15316;
TOTALIZADOR3_TON_DS5 := TOTALIZADOR3_KG_DS5 / 1000;

//Velocidade atual do dosador
%QW10316 := %IW15268;
%QW10318 := %IW15266;

VELOCIDADE_REAL_DS5 := VELOCIDADE_REAL2_DS5 ;

END_PROGRAM

